C05358=1027.695,418.842,-151.802,174.340,48.612,159.982
C05359=1027.684,418.597,-151.753,174.327,48.608,159.979
C05360=1027.673,418.352,-151.706,174.314,48.605,159.976
C05361=1027.662,418.107,-151.658,174.301,48.601,159.973
C05362=1027.651,417.862,-151.609,174.288,48.597,159.971
C05363=1027.639,417.616,-151.562,174.275,48.593,159.967
C05364=1027.628,417.372,-151.514,174.262,48.590,159.965
C05365=1027.617,417.126,-151.467,174.249,48.586,159.962
C05366=1027.606,416.881,-151.418,174.236,48.583,159.959
C05367=1027.595,416.636,-151.370,174.223,48.579,159.956
C05368=1027.584,416.390,-151.323,174.210,48.576,159.953
C05369=1027.573,416.145,-151.275,174.197,48.572,159.950
C05370=1027.562,415.900,-151.229,174.184,48.569,159.947
C05371=1027.550,415.655,-151.181,174.171,48.565,159.944
C05372=1027.539,415.409,-151.133,174.160,48.562,159.942
C05373=1027.528,415.164,-151.087,174.147,48.558,159.939
C05374=1027.517,414.918,-151.040,174.134,48.555,159.936
C05375=1027.506,414.674,-150.992,174.121,48.551,159.933
C05376=1027.495,414.428,-150.945,174.108,48.548,159.930
C05377=1027.484,414.183,-150.898,174.097,48.545,159.928
C05378=1027.473,413.937,-150.851,174.084,48.541,159.925
C05379=1027.462,413.692,-150.804,174.071,48.538,159.922
C05380=1027.450,413.446,-150.757,174.060,48.535,159.919
C05381=1027.440,413.201,-150.710,174.047,48.531,159.917
C05382=1027.429,412.956,-150.663,174.034,48.528,159.914
C05383=1027.418,412.711,-150.616,174.022,48.524,159.911
C05384=1027.407,412.465,-150.569,174.010,48.522,159.908
C05385=1027.397,412.220,-150.523,173.998,48.518,159.906
C05386=1027.386,411.975,-150.476,173.986,48.515,159.903
C05387=1027.376,411.729,-150.429,173.974,48.512,159.900
C05388=1027.364,411.484,-150.382,173.962,48.509,159.898
C05389=1027.354,411.238,-150.336,173.950,48.505,159.895
C05390=1027.343,410.993,-150.289,173.937,48.502,159.892
C05391=1027.333,410.747,-150.243,173.926,48.499,159.890
C05392=1027.322,410.502,-150.197,173.913,48.496,159.887
C05393=1027.309,410.210,-150.141,173.899,48.492,159.884
C05394=1027.297,409.918,-150.086,173.885,48.488,159.881
C05395=1027.284,409.626,-150.031,173.871,48.484,159.878
C05396=1027.271,409.334,-149.976,173.857,48.481,159.875
C05397=1027.261,409.088,-149.930,173.846,48.478,159.872
C05398=1027.250,408.842,-149.884,173.834,48.475,159.870
C05399=1027.240,408.597,-149.838,173.822,48.472,159.867
C05400=1027.229,408.351,-149.792,173.810,48.469,159.865
C05401=1027.218,408.106,-149.746,173.799,48.466,159.862
C05402=1027.208,407.860,-149.700,173.788,48.463,159.860
C05403=1027.197,407.615,-149.655,173.775,48.460,159.857
C05404=1027.186,407.370,-149.610,173.764,48.458,159.855
C05405=1027.176,407.124,-149.564,173.753,48.454,159.852
C05406=1027.165,406.879,-149.518,173.742,48.452,159.850
C05407=1027.155,406.632,-149.473,173.729,48.449,159.847
C05408=1027.145,406.387,-149.427,173.718,48.446,159.845
C05409=1027.134,406.142,-149.381,173.707,48.443,159.843
C05410=1027.123,405.896,-149.335,173.696,48.440,159.840
C05411=1027.113,405.650,-149.290,173.684,48.437,159.838
C05412=1027.103,405.405,-149.244,173.673,48.434,159.835
C05413=1027.093,405.159,-149.199,173.662,48.432,159.833
C05414=1027.083,404.914,-149.154,173.651,48.429,159.831
C05415=1027.072,404.668,-149.109,173.640,48.426,159.828
C05416=1027.062,404.422,-149.063,173.629,48.423,159.826
C05417=1027.052,404.177,-149.018,173.618,48.421,159.824
C05418=1027.042,403.931,-148.972,173.607,48.418,159.821
C05419=1027.032,403.686,-148.927,173.595,48.415,159.819
C05420=1027.021,403.439,-148.882,173.584,48.413,159.817
C05421=1027.012,403.194,-148.837,173.573,48.410,159.814
C05422=1027.002,402.949,-148.792,173.562,48.407,159.812
C05423=1026.991,402.703,-148.746,173.551,48.404,159.810
C05424=1026.982,402.457,-148.702,173.540,48.402,159.807
C05425=1026.972,402.212,-148.657,173.529,48.399,159.805
C05426=1026.962,401.966,-148.612,173.518,48.397,159.803
C05427=1026.952,401.720,-148.567,173.508,48.394,159.801
C05428=1026.942,401.475,-148.522,173.497,48.391,159.798
C05429=1026.931,401.229,-148.477,173.486,48.389,159.796
C05430=1026.921,400.983,-148.432,173.475,48.386,159.794
C05431=1026.912,400.738,-148.388,173.465,48.384,159.792
C05432=1026.902,400.492,-148.343,173.453,48.381,159.789
C05433=1026.892,400.246,-148.298,173.444,48.379,159.787
C05434=1026.882,400.000,-148.254,173.433,48.376,159.785
C05435=1026.872,399.755,-148.209,173.422,48.374,159.783
C05436=1026.862,399.509,-148.164,173.411,48.372,159.781
C05437=1026.853,399.263,-148.120,173.401,48.369,159.778
C05438=1026.842,399.018,-148.076,173.390,48.367,159.776
C05439=1026.833,398.772,-148.032,173.379,48.364,159.774
C05440=1026.823,398.525,-147.987,173.370,48.362,159.772
C05441=1026.812,398.280,-147.943,173.359,48.360,159.770
C05442=1026.803,398.034,-147.898,173.348,48.357,159.768
C05443=1026.793,397.788,-147.855,173.338,48.355,159.765
C05444=1026.783,397.542,-147.811,173.328,48.353,159.763
C05445=1026.774,397.296,-147.767,173.317,48.350,159.761
C05446=1026.763,397.051,-147.723,173.307,48.348,159.759
C05447=1026.754,396.805,-147.678,173.296,48.346,159.757
C05448=1026.744,396.559,-147.635,173.287,48.343,159.755
C05449=1026.734,396.313,-147.591,173.276,48.342,159.753
C05450=1026.724,396.067,-147.547,173.266,48.339,159.751
C05451=1026.715,395.821,-147.504,173.256,48.337,159.749
C05452=1026.705,395.576,-147.460,173.246,48.334,159.747
C05453=1026.695,395.306,-147.412,173.234,48.332,159.744
C05454=1026.684,395.034,-147.363,173.223,48.330,159.742
C05455=1026.674,394.765,-147.315,173.212,48.327,159.740
C05456=1026.663,394.495,-147.267,173.202,48.325,159.738
C05457=1026.653,394.249,-147.224,173.191,48.323,159.736
C05458=1026.645,394.003,-147.180,173.181,48.321,159.734
C05459=1026.634,393.757,-147.137,173.171,48.319,159.732
C05460=1026.625,393.511,-147.093,173.161,48.317,159.730
C05461=1026.615,393.265,-147.050,173.152,48.315,159.728
C05462=1026.606,393.019,-147.006,173.141,48.312,159.726
C05463=1026.597,392.773,-146.963,173.132,48.310,159.724
C05464=1026.586,392.527,-146.920,173.121,48.309,159.722
C05465=1026.578,392.281,-146.877,173.112,48.307,159.720
C05466=1026.568,392.035,-146.833,173.102,48.304,159.718
C05467=1026.558,391.789,-146.791,173.092,48.303,159.716
C05468=1026.549,391.543,-146.747,173.082,48.301,159.714
C05469=1026.539,391.297,-146.704,173.073,48.299,159.712
C05470=1026.530,391.051,-146.662,173.063,48.297,159.711
C05471=1026.521,390.805,-146.618,173.053,48.295,159.709
C05472=1026.511,390.559,-146.575,173.044,48.293,159.707
C05473=1026.502,390.312,-146.532,173.034,48.291,159.705
C05474=1026.493,390.067,-146.489,173.024,48.289,159.703
C05475=1026.483,389.821,-146.446,173.014,48.287,159.701
C05476=1026.474,389.575,-146.403,173.005,48.285,159.699
C05477=1026.465,389.329,-146.360,172.996,48.283,159.697
C05478=1026.455,389.083,-146.317,172.987,48.282,159.696
C05479=1026.446,388.837,-146.275,172.976,48.280,159.694
C05480=1026.437,388.590,-146.232,172.967,48.278,159.692
C05481=1026.428,388.344,-146.189,172.957,48.276,159.690
C05482=1026.418,388.097,-146.147,172.948,48.275,159.688
C05483=1026.409,387.852,-146.105,172.939,48.273,159.686
C05484=1026.400,387.606,-146.062,172.930,48.271,159.685
C05485=1026.391,387.360,-146.019,172.920,48.269,159.683
C05486=1026.381,387.113,-145.976,172.910,48.268,159.681
C05487=1026.372,386.867,-145.935,172.901,48.266,159.679
C05488=1026.363,386.621,-145.892,172.892,48.264,159.677
C05489=1026.354,386.376,-145.850,172.883,48.263,159.676
C05490=1026.344,386.128,-145.808,172.873,48.261,159.674
C05491=1026.335,385.883,-145.765,172.864,48.259,159.672
C05492=1026.326,385.636,-145.724,172.855,48.258,159.671
C05493=1026.317,385.391,-145.681,172.846,48.256,159.669
C05494=1026.307,385.144,-145.639,172.837,48.255,159.667
C05495=1026.299,384.897,-145.597,172.828,48.253,159.665
C05496=1026.289,384.651,-145.555,172.818,48.252,159.664
C05497=1026.280,384.405,-145.513,172.809,48.250,159.662
C05498=1026.271,384.159,-145.472,172.800,48.248,159.660
C05499=1026.262,383.913,-145.429,172.791,48.247,159.659
C05500=1026.253,383.667,-145.387,172.782,48.245,159.657
C05501=1026.244,383.420,-145.346,172.773,48.244,159.655
C05502=1026.235,383.174,-145.304,172.764,48.242,159.654
C05503=1026.226,382.927,-145.262,172.755,48.241,159.652
C05504=1026.218,382.681,-145.221,172.746,48.240,159.650
C05505=1026.209,382.435,-145.179,172.737,48.238,159.649
C05506=1026.199,382.189,-145.138,172.728,48.237,159.647
C05507=1026.190,381.942,-145.096,172.719,48.235,159.645
C05508=1026.181,381.696,-145.054,172.710,48.234,159.644
C05509=1026.172,381.456,-145.013,172.702,48.233,159.642
C05510=1026.163,381.216,-144.972,172.693,48.231,159.641
C05511=1026.155,380.976,-144.932,172.684,48.230,159.639
C05512=1026.146,380.736,-144.891,172.676,48.229,159.638
C05513=1026.138,380.496,-144.851,172.667,48.227,159.636
C05514=1026.129,380.257,-144.811,172.659,48.226,159.634
C05515=1026.120,380.017,-144.770,172.650,48.225,159.633
C05516=1026.112,379.776,-144.730,172.641,48.223,159.631
C05517=1026.104,379.530,-144.689,172.632,48.222,159.630
C05518=1026.095,379.284,-144.647,172.624,48.220,159.628
C05519=1026.086,379.037,-144.606,172.616,48.220,159.627
C05520=1026.077,378.790,-144.565,172.607,48.218,159.625
C05521=1026.068,378.545,-144.524,172.598,48.217,159.623
C05522=1026.059,378.298,-144.483,172.590,48.216,159.622
C05523=1026.051,378.052,-144.441,172.581,48.214,159.620
C05524=1026.042,377.805,-144.400,172.572,48.213,159.619
C05525=1026.034,377.559,-144.359,172.564,48.212,159.617
C05526=1026.025,377.312,-144.318,172.555,48.211,159.616
C05527=1026.017,377.066,-144.276,172.547,48.210,159.614
C05528=1026.008,376.819,-144.235,172.539,48.208,159.613
C05529=1025.999,376.573,-144.195,172.530,48.207,159.611
C05530=1025.990,376.327,-144.154,172.521,48.206,159.610
C05531=1025.982,376.080,-144.113,172.512,48.205,159.608
C05532=1025.972,375.833,-144.072,172.505,48.204,159.607
C05533=1025.964,375.587,-144.032,172.496,48.203,159.605
C05534=1025.955,375.340,-143.991,172.488,48.201,159.604
C05535=1025.947,375.094,-143.951,172.479,48.201,159.602
C05536=1025.937,374.847,-143.910,172.470,48.200,159.601
C05537=1025.929,374.601,-143.869,172.463,48.199,159.600
C05538=1025.921,374.354,-143.828,172.454,48.198,159.598
C05539=1025.912,374.108,-143.788,172.445,48.197,159.597
C05540=1025.903,373.861,-143.747,172.438,48.196,159.595
C05541=1025.895,373.615,-143.707,172.429,48.195,159.594
C05542=1025.886,373.368,-143.666,172.421,48.193,159.592
C05543=1025.877,373.122,-143.626,172.413,48.193,159.591
C05544=1025.869,372.875,-143.585,172.405,48.191,159.589
C05545=1025.861,372.628,-143.545,172.396,48.191,159.588
C05546=1025.852,372.382,-143.505,172.388,48.190,159.587
C05547=1025.844,372.135,-143.464,172.380,48.189,159.585
C05548=1025.835,371.889,-143.424,172.371,48.188,159.584
C05549=1025.827,371.642,-143.384,172.364,48.187,159.583
C05550=1025.818,371.396,-143.344,172.355,48.187,159.581
C05551=1025.810,371.149,-143.303,172.348,48.185,159.580
C05552=1025.802,370.903,-143.263,172.340,48.184,159.578
C05553=1025.793,370.656,-143.223,172.331,48.184,159.577
C05554=1025.785,370.409,-143.183,172.324,48.183,159.576
C05555=1025.776,370.163,-143.143,172.315,48.182,159.574
C05556=1025.768,369.916,-143.103,172.308,48.181,159.573
C05557=1025.760,369.670,-143.063,172.299,48.180,159.572
C05558=1025.751,369.423,-143.023,172.292,48.180,159.571
C05559=1025.743,369.176,-142.982,172.283,48.179,159.569
C05560=1025.735,368.930,-142.943,172.276,48.178,159.568
C05561=1025.727,368.683,-142.903,172.268,48.177,159.566
C05562=1025.718,368.437,-142.863,172.259,48.177,159.565
C05563=1025.710,368.190,-142.824,172.252,48.176,159.564
C05564=1025.701,367.943,-142.784,172.243,48.175,159.563
C05565=1025.693,367.696,-142.744,172.236,48.175,159.561
C05566=1025.685,367.449,-142.705,172.228,48.173,159.560
C05567=1025.676,367.203,-142.665,172.220,48.173,159.559
C05568=1025.668,366.956,-142.626,172.213,48.173,159.558
C05569=1025.660,366.727,-142.589,172.205,48.172,159.556
C05570=1025.652,366.498,-142.552,172.198,48.171,159.555
C05571=1025.645,366.269,-142.515,172.190,48.171,159.554
C05572=1025.637,366.039,-142.479,172.183,48.170,159.553
C05573=1025.629,365.809,-142.442,172.176,48.170,159.552
C05574=1025.622,365.580,-142.405,172.169,48.170,159.551
C05575=1025.614,365.351,-142.369,172.162,48.169,159.549
C05576=1025.607,365.122,-142.332,172.155,48.168,159.548
C05577=1025.598,364.875,-142.293,172.147,48.168,159.547
C05578=1025.590,364.629,-142.253,172.139,48.167,159.546
C05579=1025.582,364.381,-142.215,172.132,48.166,159.545
C05580=1025.573,364.135,-142.175,172.124,48.166,159.543
C05581=1025.566,363.888,-142.136,172.116,48.166,159.542
C05582=1025.557,363.641,-142.096,172.109,48.165,159.541
C05583=1025.549,363.394,-142.058,172.101,48.164,159.540
C05584=1025.540,363.147,-142.018,172.094,48.164,159.539
C05585=1025.533,362.901,-141.978,172.086,48.163,159.537
C05586=1025.525,362.654,-141.940,172.079,48.163,159.536
C05587=1025.517,362.407,-141.901,172.071,48.163,159.535
C05588=1025.509,362.160,-141.862,172.064,48.162,159.534
C05589=1025.500,361.914,-141.823,172.056,48.161,159.533
C05590=1025.493,361.666,-141.784,172.048,48.161,159.531
C05591=1025.485,361.420,-141.745,172.041,48.161,159.530
C05592=1025.477,361.173,-141.706,172.034,48.160,159.529
C05593=1025.468,360.926,-141.667,172.026,48.160,159.528
C05594=1025.460,360.679,-141.628,172.019,48.159,159.527
C05595=1025.453,360.433,-141.589,172.012,48.159,159.526
C05596=1025.445,360.186,-141.550,172.004,48.159,159.525
C05597=1025.437,359.939,-141.511,171.997,48.159,159.524
C05598=1025.428,359.691,-141.473,171.989,48.158,159.522
C05599=1025.421,359.445,-141.434,171.982,48.158,159.521
C05600=1025.412,359.198,-141.395,171.975,48.158,159.520
C05601=1025.404,358.951,-141.357,171.968,48.158,159.519
C05602=1025.397,358.705,-141.318,171.959,48.157,159.518
C05603=1025.388,358.458,-141.280,171.952,48.157,159.517
C05604=1025.380,358.210,-141.242,171.945,48.157,159.516
C05605=1025.372,357.964,-141.204,171.938,48.157,159.515
C05606=1025.364,357.717,-141.165,171.931,48.157,159.514
C05607=1025.356,357.470,-141.127,171.924,48.156,159.513
C05608=1025.348,357.223,-141.088,171.916,48.156,159.512
C05609=1025.340,356.976,-141.049,171.909,48.156,159.511
C05610=1025.333,356.729,-141.011,171.902,48.155,159.509
C05611=1025.324,356.482,-140.973,171.895,48.155,159.508
C05612=1025.317,356.235,-140.934,171.888,48.155,159.507
C05613=1025.308,355.989,-140.896,171.880,48.155,159.506
C05614=1025.301,355.741,-140.859,171.873,48.155,159.505
C05615=1025.293,355.494,-140.820,171.866,48.155,159.504
C05616=1025.285,355.248,-140.782,171.859,48.155,159.503
C05617=1025.277,355.000,-140.743,171.852,48.155,159.502
C05618=1025.270,354.753,-140.706,171.844,48.155,159.501
C05619=1025.262,354.506,-140.667,171.837,48.155,159.500
C05620=1025.253,354.260,-140.630,171.830,48.155,159.499
C05621=1025.246,354.013,-140.592,171.823,48.155,159.498
C05622=1025.238,353.766,-140.553,171.816,48.155,159.497
C05623=1025.230,353.519,-140.516,171.809,48.155,159.496
C05624=1025.222,353.272,-140.478,171.802,48.155,159.495
C05625=1025.214,353.024,-140.440,171.795,48.154,159.494
C05626=1025.206,352.778,-140.403,171.788,48.154,159.493
C05627=1025.198,352.530,-140.365,171.781,48.154,159.492
C05628=1025.191,352.284,-140.327,171.774,48.154,159.491
C05629=1025.183,352.058,-140.292,171.768,48.155,159.490
C05630=1025.176,351.832,-140.258,171.761,48.155,159.489
C05631=1025.170,351.606,-140.223,171.755,48.154,159.488
C05632=1025.162,351.380,-140.189,171.749,48.155,159.488
C05633=1025.155,351.154,-140.154,171.743,48.155,159.487
C05634=1025.147,350.928,-140.120,171.737,48.155,159.486
C05635=1025.141,350.702,-140.086,171.730,48.155,159.485
C05636=1025.134,350.476,-140.051,171.724,48.155,159.484
C05637=1025.126,350.229,-140.014,171.717,48.155,159.483
C05638=1025.119,349.982,-139.976,171.710,48.155,159.482
C05639=1025.111,349.734,-139.939,171.704,48.156,159.481
C05640=1025.103,349.488,-139.901,171.696,48.156,159.480
C05641=1025.096,349.241,-139.863,171.689,48.155,159.479
C05642=1025.088,348.993,-139.826,171.683,48.156,159.479
C05643=1025.080,348.747,-139.789,171.676,48.156,159.478
C05644=1025.073,348.499,-139.751,171.670,48.156,159.477
C05645=1025.065,348.252,-139.714,171.663,48.156,159.476
C05646=1025.057,348.005,-139.677,171.656,48.156,159.475
C05647=1025.050,347.758,-139.639,171.649,48.157,159.474
C05648=1025.042,347.511,-139.602,171.642,48.157,159.473
C05649=1025.035,347.264,-139.565,171.636,48.157,159.472
C05650=1025.027,347.017,-139.528,171.629,48.158,159.471
C05651=1025.019,346.769,-139.491,171.622,48.158,159.470
C05652=1025.012,346.522,-139.454,171.616,48.158,159.470
C05653=1025.004,346.275,-139.417,171.609,48.158,159.469
C05654=1024.997,346.028,-139.379,171.602,48.159,159.468
C05655=1024.988,345.781,-139.342,171.596,48.159,159.467
C05656=1024.981,345.533,-139.305,171.589,48.159,159.466
C05657=1024.973,345.286,-139.268,171.582,48.160,159.465
C05658=1024.965,345.039,-139.232,171.576,48.160,159.465
C05659=1024.958,344.792,-139.195,171.570,48.161,159.464
C05660=1024.950,344.545,-139.158,171.562,48.161,159.463
C05661=1024.943,344.297,-139.121,171.556,48.161,159.462
C05662=1024.936,344.051,-139.084,171.549,48.162,159.461
C05663=1024.928,343.804,-139.047,171.543,48.162,159.460
C05664=1024.921,343.556,-139.011,171.537,48.163,159.460
C05665=1024.913,343.310,-138.974,171.530,48.162,159.459
C05666=1024.905,343.062,-138.937,171.523,48.163,159.458
C05667=1024.898,342.815,-138.900,171.517,48.163,159.457
C05668=1024.890,342.567,-138.864,171.511,48.164,159.456
C05669=1024.883,342.320,-138.828,171.504,48.164,159.455
C05670=1024.876,342.073,-138.790,171.497,48.165,159.455
C05671=1024.868,341.825,-138.754,171.491,48.165,159.454
C05672=1024.860,341.579,-138.717,171.485,48.166,159.453
C05673=1024.854,341.332,-138.680,171.478,48.166,159.452
C05674=1024.846,341.084,-138.644,171.471,48.167,159.451
C05675=1024.838,340.837,-138.608,171.466,48.167,159.451
C05676=1024.831,340.590,-138.570,171.459,48.168,159.450
C05677=1024.824,340.343,-138.535,171.452,48.168,159.449
C05678=1024.816,340.095,-138.498,171.446,48.169,159.448
C05679=1024.809,339.848,-138.462,171.440,48.169,159.448
C05680=1024.802,339.600,-138.425,171.433,48.170,159.447
C05681=1024.794,339.353,-138.388,171.427,48.171,159.446
C05682=1024.787,339.107,-138.353,171.421,48.171,159.445
C05683=1024.779,338.859,-138.316,171.414,48.172,159.445
C05684=1024.771,338.612,-138.280,171.408,48.172,159.444
C05685=1024.764,338.365,-138.244,171.401,48.173,159.443
C05686=1024.756,338.118,-138.208,171.396,48.174,159.442
C05687=1024.749,337.870,-138.172,171.389,48.174,159.442
C05688=1024.741,337.622,-138.136,171.383,48.176,159.441
C05689=1024.735,337.395,-138.102,171.377,48.176,159.440
C05690=1024.728,337.168,-138.070,171.372,48.177,159.440
C05691=1024.721,336.940,-138.036,171.366,48.177,159.439
C05692=1024.714,336.713,-138.003,171.359,48.178,159.438
C05693=1024.708,336.485,-137.970,171.354,48.178,159.438
C05694=1024.700,336.257,-137.937,171.348,48.179,159.437
C05695=1024.694,336.030,-137.904,171.343,48.179,159.436
C05696=1024.687,335.803,-137.871,171.337,48.180,159.436
C05697=1024.680,335.555,-137.836,171.331,48.181,159.435
C05698=1024.673,335.307,-137.799,171.324,48.182,159.434
C05699=1024.666,335.061,-137.763,171.319,48.182,159.434
C05700=1024.658,334.813,-137.727,171.312,48.184,159.433
C05701=1024.651,334.565,-137.691,171.306,48.184,159.432
C05702=1024.644,334.318,-137.656,171.300,48.185,159.432
C05703=1024.636,334.071,-137.619,171.293,48.186,159.431
C05704=1024.629,333.824,-137.584,171.288,48.186,159.430
C05705=1024.622,333.576,-137.548,171.281,48.187,159.429
C05706=1024.615,333.329,-137.513,171.275,48.188,159.429
C05707=1024.607,333.081,-137.477,171.270,48.189,159.428
C05708=1024.600,332.834,-137.442,171.263,48.190,159.427
C05709=1024.592,332.587,-137.406,171.258,48.190,159.427
C05710=1024.585,332.340,-137.371,171.251,48.192,159.426
C05711=1024.578,332.093,-137.335,171.245,48.193,159.426
C05712=1024.571,331.845,-137.299,171.239,48.193,159.425
C05713=1024.563,331.598,-137.265,171.233,48.194,159.424
C05714=1024.556,331.350,-137.229,171.227,48.195,159.424
C05715=1024.549,331.103,-137.194,171.221,48.196,159.423
C05716=1024.542,330.855,-137.158,171.215,48.198,159.423
C05717=1024.535,330.607,-137.123,171.209,48.198,159.422
C05718=1024.527,330.361,-137.088,171.203,48.199,159.421
C05719=1024.520,330.113,-137.052,171.197,48.200,159.421
C05720=1024.513,329.866,-137.017,171.191,48.201,159.420
C05721=1024.506,329.618,-136.982,171.185,48.202,159.419
C05722=1024.498,329.371,-136.946,171.179,48.203,159.419
C05723=1024.491,329.124,-136.911,171.174,48.204,159.418
C05724=1024.484,328.876,-136.876,171.167,48.205,159.418
C05725=1024.477,328.628,-136.840,171.161,48.206,159.417
C05726=1024.470,328.381,-136.805,171.156,48.207,159.416
C05727=1024.463,328.134,-136.771,171.149,48.208,159.416
C05728=1024.456,327.886,-136.736,171.144,48.209,159.415
C05729=1024.448,327.638,-136.700,171.138,48.210,159.415
C05730=1024.441,327.392,-136.664,171.132,48.211,159.414
C05731=1024.435,327.144,-136.629,171.126,48.212,159.414
C05732=1024.427,326.897,-136.595,171.120,48.213,159.413
C05733=1024.419,326.649,-136.560,171.114,48.215,159.412
C05734=1024.412,326.401,-136.525,171.109,48.215,159.412
C05735=1024.405,326.154,-136.491,171.103,48.217,159.411
C05736=1024.397,325.907,-136.456,171.097,48.218,159.411
C05737=1024.390,325.659,-136.421,171.091,48.219,159.410
C05738=1024.383,325.412,-136.387,171.085,48.220,159.410
C05739=1024.375,325.165,-136.352,171.079,48.222,159.409
C05740=1024.369,324.917,-136.318,171.073,48.223,159.409
C05741=1024.361,324.670,-136.283,171.068,48.224,159.408
C05742=1024.353,324.422,-136.248,171.062,48.226,159.408
C05743=1024.347,324.174,-136.214,171.056,48.227,159.407
C05744=1024.339,323.927,-136.180,171.050,48.228,159.406
C05745=1024.332,323.680,-136.145,171.045,48.229,159.406
C05746=1024.325,323.432,-136.111,171.039,48.231,159.405
C05747=1024.318,323.185,-136.076,171.034,48.232,159.405
C05748=1024.311,322.937,-136.042,171.027,48.233,159.404
C05749=1024.304,322.707,-136.010,171.022,48.235,159.404
C05750=1024.297,322.477,-135.977,171.017,48.236,159.404
C05751=1024.290,322.248,-135.946,171.011,48.237,159.403
C05752=1024.284,322.018,-135.914,171.006,48.238,159.403
C05753=1024.277,321.788,-135.881,171.001,48.240,159.402
C05754=1024.270,321.558,-135.850,170.996,48.240,159.402
C05755=1024.264,321.328,-135.818,170.991,48.242,159.401
C05756=1024.258,321.099,-135.786,170.986,48.243,159.401
C05757=1024.251,320.851,-135.752,170.980,48.245,159.400
C05758=1024.243,320.604,-135.718,170.974,48.245,159.400
C05759=1024.236,320.356,-135.684,170.968,48.247,159.399
C05760=1024.230,320.108,-135.649,170.963,48.248,159.399
C05761=1024.222,319.861,-135.615,170.957,48.250,159.398
C05762=1024.215,319.614,-135.581,170.952,48.251,159.398
C05763=1024.208,319.366,-135.547,170.946,48.252,159.397
C05764=1024.201,319.118,-135.512,170.940,48.254,159.397
C05765=1024.194,318.871,-135.478,170.935,48.256,159.397
C05766=1024.187,318.623,-135.444,170.929,48.257,159.396
C05767=1024.180,318.375,-135.410,170.924,48.258,159.396
C05768=1024.173,318.129,-135.376,170.918,48.260,159.395
C05769=1024.167,317.881,-135.341,170.912,48.261,159.395
C05770=1024.160,317.633,-135.307,170.907,48.263,159.394
C05771=1024.152,317.385,-135.274,170.901,48.264,159.394
C05772=1024.146,317.137,-135.239,170.896,48.265,159.393
C05773=1024.138,316.890,-135.205,170.890,48.267,159.393
C05774=1024.132,316.643,-135.171,170.885,48.269,159.393
C05775=1024.125,316.396,-135.137,170.880,48.270,159.392
C05776=1024.118,316.148,-135.103,170.874,48.271,159.392
C05777=1024.111,315.900,-135.069,170.868,48.273,159.391
C05778=1024.104,315.652,-135.035,170.863,48.274,159.391
C05779=1024.098,315.405,-135.001,170.857,48.276,159.390
C05780=1024.091,315.157,-134.967,170.852,48.278,159.390
C05781=1024.083,314.910,-134.934,170.846,48.279,159.390
C05782=1024.077,314.662,-134.899,170.841,48.281,159.389
C05783=1024.070,314.415,-134.866,170.836,48.282,159.389
C05784=1024.063,314.167,-134.832,170.830,48.284,159.388
C05785=1024.056,313.919,-134.798,170.825,48.285,159.388
C05786=1024.050,313.672,-134.764,170.820,48.287,159.387
C05787=1024.043,313.425,-134.730,170.814,48.288,159.387
C05788=1024.036,313.177,-134.696,170.809,48.290,159.387
C05789=1024.030,312.930,-134.662,170.804,48.291,159.386
C05790=1024.023,312.681,-134.629,170.798,48.293,159.386
C05791=1024.016,312.434,-134.596,170.793,48.295,159.385
C05792=1024.009,312.187,-134.562,170.788,48.296,159.385
C05793=1024.003,311.939,-134.528,170.783,48.298,159.385
C05794=1023.996,311.692,-134.494,170.777,48.299,159.384
C05795=1023.989,311.444,-134.460,170.771,48.301,159.384
C05796=1023.983,311.196,-134.428,170.766,48.302,159.384
C05797=1023.976,310.948,-134.393,170.760,48.304,159.383
C05798=1023.970,310.701,-134.360,170.755,48.306,159.383
C05799=1023.962,310.454,-134.326,170.750,48.307,159.382
C05800=1023.955,310.205,-134.293,170.744,48.309,159.382
C05801=1023.949,309.958,-134.260,170.740,48.311,159.382
C05802=1023.941,309.711,-134.227,170.735,48.313,159.381
C05803=1023.935,309.463,-134.194,170.728,48.315,159.381
C05804=1023.928,309.215,-134.160,170.724,48.317,159.381
C05805=1023.920,308.967,-134.128,170.718,48.319,159.380
C05806=1023.914,308.720,-134.095,170.713,48.321,159.380
C05807=1023.907,308.472,-134.061,170.708,48.322,159.380
C05808=1023.900,308.225,-134.029,170.702,48.324,159.379
C05809=1023.893,307.997,-133.999,170.697,48.326,159.379
C05810=1023.886,307.770,-133.968,170.693,48.327,159.379
C05811=1023.880,307.543,-133.938,170.689,48.330,159.379
C05812=1023.874,307.316,-133.908,170.684,48.331,159.378
C05813=1023.868,307.089,-133.878,170.678,48.333,159.378
C05814=1023.861,306.861,-133.848,170.674,48.335,159.378
C05815=1023.855,306.634,-133.817,170.669,48.336,159.377
C05816=1023.849,306.407,-133.787,170.664,48.338,159.377
C05817=1023.842,306.159,-133.754,170.659,48.340,159.377
C05818=1023.835,305.911,-133.722,170.654,48.342,159.377
C05819=1023.827,305.664,-133.688,170.648,48.344,159.376
C05820=1023.821,305.416,-133.655,170.644,48.346,159.376
C05821=1023.814,305.169,-133.623,170.639,48.347,159.376
C05822=1023.807,304.921,-133.590,170.633,48.350,159.375
C05823=1023.801,304.673,-133.557,170.628,48.352,159.375
C05824=1023.793,304.425,-133.525,170.623,48.354,159.375
C05825=1023.787,304.177,-133.492,170.617,48.356,159.375
C05826=1023.781,303.930,-133.459,170.612,48.357,159.374
C05827=1023.773,303.682,-133.427,170.608,48.360,159.374
C05828=1023.767,303.434,-133.394,170.602,48.362,159.374
C05829=1023.760,303.186,-133.361,170.597,48.364,159.373
C05830=1023.753,302.939,-133.329,170.592,48.366,159.373
C05831=1023.747,302.691,-133.296,170.587,48.368,159.373
C05832=1023.740,302.444,-133.264,170.581,48.370,159.373
C05833=1023.733,302.195,-133.231,170.577,48.372,159.372
C05834=1023.726,301.948,-133.198,170.572,48.374,159.372
C05835=1023.719,301.701,-133.166,170.567,48.376,159.372
C05836=1023.712,301.452,-133.133,170.561,48.378,159.372
C05837=1023.706,301.205,-133.100,170.557,48.380,159.371
C05838=1023.699,300.957,-133.068,170.552,48.382,159.371
C05839=1023.692,300.709,-133.035,170.547,48.384,159.371
C05840=1023.685,300.461,-133.003,170.541,48.386,159.371
C05841=1023.679,300.214,-132.971,170.536,48.388,159.370
C05842=1023.673,299.966,-132.938,170.532,48.391,159.370
C05843=1023.666,299.719,-132.906,170.527,48.393,159.370
C05844=1023.659,299.470,-132.873,170.521,48.394,159.370
C05845=1023.653,299.222,-132.841,170.516,48.397,159.369
C05846=1023.646,298.975,-132.809,170.512,48.399,159.369
C05847=1023.640,298.727,-132.776,170.507,48.401,159.369
C05848=1023.633,298.480,-132.744,170.501,48.403,159.369
C05849=1023.626,298.231,-132.711,170.496,48.406,159.369
C05850=1023.620,297.984,-132.679,170.492,48.408,159.368
C05851=1023.613,297.736,-132.646,170.487,48.409,159.368
C05852=1023.607,297.488,-132.614,170.482,48.411,159.368
C05853=1023.600,297.241,-132.582,170.476,48.414,159.368
C05854=1023.593,296.993,-132.549,170.472,48.416,159.367
C05855=1023.587,296.745,-132.517,170.467,48.418,159.367
C05856=1023.580,296.498,-132.485,170.462,48.420,159.367
C05857=1023.574,296.249,-132.453,170.458,48.422,159.367
C05858=1023.567,296.001,-132.420,170.452,48.425,159.367
C05859=1023.561,295.753,-132.389,170.447,48.427,159.366
C05860=1023.554,295.506,-132.356,170.442,48.429,159.366
C05861=1023.547,295.258,-132.324,170.438,48.431,159.366
C05862=1023.541,295.010,-132.292,170.433,48.433,159.366
C05863=1023.535,294.763,-132.259,170.427,48.436,159.366
C05864=1023.528,294.515,-132.228,170.423,48.438,159.365
C05865=1023.522,294.267,-132.196,170.418,48.440,159.365
C05866=1023.515,294.019,-132.163,170.413,48.442,159.365
C05867=1023.509,293.771,-132.131,170.408,48.445,159.365
C05868=1023.502,293.524,-132.099,170.404,48.447,159.365
C05869=1023.497,293.305,-132.071,170.399,48.450,159.365
C05870=1023.491,293.086,-132.043,170.395,48.452,159.365
C05871=1023.485,292.868,-132.015,170.391,48.454,159.364
C05872=1023.480,292.650,-131.987,170.386,48.456,159.364
C05873=1023.473,292.430,-131.959,170.383,48.458,159.364
C05874=1023.467,292.212,-131.931,170.378,48.460,159.364
C05875=1023.462,291.994,-131.903,170.373,48.462,159.364
C05876=1023.456,291.775,-131.876,170.370,48.464,159.364
C05877=1023.450,291.527,-131.844,170.365,48.467,159.364
C05878=1023.443,291.280,-131.812,170.359,48.469,159.363
C05879=1023.437,291.032,-131.780,170.355,48.471,159.363
C05880=1023.430,290.784,-131.749,170.350,48.474,159.363
C05881=1023.423,290.536,-131.717,170.346,48.476,159.363
C05882=1023.416,290.288,-131.686,170.341,48.478,159.363
C05883=1023.410,290.040,-131.654,170.336,48.481,159.363
C05884=1023.403,289.792,-131.623,170.331,48.483,159.363
C05885=1023.396,289.545,-131.591,170.327,48.486,159.363
C05886=1023.390,289.297,-131.560,170.322,48.488,159.362
C05887=1023.384,289.048,-131.528,170.317,48.491,159.362
C05888=1023.377,288.801,-131.497,170.312,48.494,159.362
C05889=1023.370,288.553,-131.465,170.307,48.497,159.362
C05890=1023.363,288.305,-131.434,170.303,48.499,159.362
C05891=1023.357,288.057,-131.402,170.298,48.501,159.362
C05892=1023.351,287.810,-131.371,170.294,48.504,159.362
C05893=1023.344,287.561,-131.341,170.288,48.507,159.362
C05894=1023.337,287.313,-131.309,170.284,48.509,159.361
C05895=1023.331,287.065,-131.278,170.279,48.512,159.361
C05896=1023.324,286.817,-131.246,170.275,48.514,159.361
C05897=1023.317,286.569,-131.215,170.270,48.517,159.361
C05898=1023.311,286.321,-131.184,170.265,48.519,159.361
C05899=1023.305,286.073,-131.152,170.260,48.522,159.361
C05900=1023.299,285.826,-131.121,170.256,48.525,159.361
C05901=1023.292,285.578,-131.090,170.251,48.527,159.361
C05902=1023.285,285.330,-131.058,170.247,48.530,159.361
C05903=1023.278,285.082,-131.028,170.242,48.533,159.361
C05904=1023.271,284.834,-130.997,170.237,48.535,159.361
C05905=1023.266,284.586,-130.966,170.232,48.538,159.361
C05906=1023.259,284.338,-130.935,170.228,48.541,159.361
C05907=1023.252,284.090,-130.903,170.223,48.543,159.361
C05908=1023.246,283.841,-130.873,170.219,48.546,159.360
C05909=1023.238,283.594,-130.842,170.214,48.548,159.360
C05910=1023.232,283.346,-130.811,170.209,48.552,159.360
C05911=1023.226,283.098,-130.780,170.205,48.554,159.360
C05912=1023.219,282.850,-130.749,170.200,48.557,159.360
C05913=1023.213,282.602,-130.718,170.196,48.559,159.360
C05914=1023.207,282.354,-130.688,170.191,48.562,159.360
C05915=1023.199,282.106,-130.657,170.186,48.565,159.360
C05916=1023.193,281.858,-130.626,170.182,48.568,159.360
C05917=1023.186,281.610,-130.595,170.177,48.571,159.360
C05918=1023.180,281.362,-130.564,170.173,48.574,159.360
C05919=1023.174,281.114,-130.533,170.168,48.576,159.360
C05920=1023.166,280.866,-130.503,170.164,48.579,159.360
C05921=1023.161,280.618,-130.472,170.158,48.582,159.360
C05922=1023.154,280.370,-130.441,170.154,48.585,159.360
C05923=1023.147,280.122,-130.410,170.150,48.587,159.360
C05924=1023.142,279.874,-130.380,170.145,48.590,159.360
C05925=1023.135,279.626,-130.348,170.141,48.593,159.360
C05926=1023.128,279.378,-130.318,170.137,48.596,159.360
C05927=1023.122,279.130,-130.288,170.132,48.599,159.360
C05928=1023.115,278.882,-130.256,170.127,48.602,159.360
C05929=1023.110,278.669,-130.230,170.123,48.604,159.360
C05930=1023.104,278.457,-130.204,170.120,48.606,159.360
C05931=1023.099,278.245,-130.178,170.115,48.609,159.360
C05932=1023.093,278.032,-130.152,170.112,48.611,159.360
C05933=1023.088,277.820,-130.125,170.108,48.614,159.360
C05934=1023.083,277.608,-130.099,170.104,48.616,159.359
C05935=1023.077,277.396,-130.073,170.101,48.619,159.360
C05936=1023.071,277.182,-130.047,170.096,48.621,159.360
C05937=1023.065,276.934,-130.016,170.092,48.624,159.360
C05938=1023.058,276.686,-129.986,170.088,48.627,159.360
C05939=1023.052,276.438,-129.956,170.083,48.630,159.360
C05940=1023.045,276.190,-129.926,170.079,48.633,159.360
C05941=1023.039,275.943,-129.895,170.074,48.637,159.360
C05942=1023.032,275.695,-129.865,170.069,48.639,159.360
C05943=1023.026,275.447,-129.834,170.065,48.642,159.360
C05944=1023.020,275.198,-129.803,170.061,48.645,159.360
C05945=1023.013,274.950,-129.773,170.056,48.648,159.360
C05946=1023.007,274.702,-129.743,170.052,48.651,159.360
C05947=1023.000,274.454,-129.713,170.047,48.654,159.360
C05948=1022.994,274.206,-129.683,170.043,48.657,159.360
C05949=1022.987,273.958,-129.653,170.038,48.660,159.360
C05950=1022.981,273.710,-129.623,170.034,48.664,159.360
C05951=1022.974,273.462,-129.593,170.030,48.666,159.360
C05952=1022.968,273.214,-129.562,170.026,48.669,159.360
C05953=1022.962,272.965,-129.532,170.021,48.672,159.360
C05954=1022.955,272.718,-129.502,170.016,48.676,159.360
C05955=1022.948,272.469,-129.472,170.012,48.679,159.360
C05956=1022.942,272.222,-129.441,170.007,48.681,159.360
C05957=1022.936,271.974,-129.412,170.003,48.685,159.360
C05958=1022.930,271.725,-129.382,169.999,48.688,159.360
C05959=1022.923,271.477,-129.352,169.995,48.691,159.360
C05960=1022.917,271.229,-129.321,169.991,48.694,159.360
C05961=1022.910,270.981,-129.291,169.985,48.697,159.360
C05962=1022.904,270.732,-129.261,169.981,48.701,159.360
C05963=1022.897,270.485,-129.232,169.977,48.703,159.360
C05964=1022.892,270.237,-129.201,169.973,48.707,159.361
C05965=1022.885,269.988,-129.172,169.969,48.710,159.361
C05966=1022.878,269.741,-129.142,169.965,48.713,159.361
C05967=1022.872,269.492,-129.111,169.960,48.716,159.361
C05968=1022.866,269.244,-129.082,169.955,48.720,159.361
C05969=1022.859,268.996,-129.053,169.951,48.723,159.361
C05970=1022.853,268.748,-129.022,169.947,48.726,159.361
C05971=1022.846,268.500,-128.993,169.942,48.729,159.361
C05972=1022.839,268.252,-128.963,169.938,48.732,159.361
C05973=1022.834,268.003,-128.933,169.934,48.735,159.361
C05974=1022.827,267.756,-128.903,169.930,48.739,159.361
C05975=1022.820,267.507,-128.874,169.925,48.743,159.361
C05976=1022.814,267.259,-128.844,169.921,48.745,159.361
C05977=1022.808,267.011,-128.815,169.917,48.749,159.362
C05978=1022.801,266.763,-128.784,169.912,48.752,159.362
C05979=1022.795,266.515,-128.755,169.908,48.755,159.362
C05980=1022.789,266.267,-128.725,169.904,48.759,159.362
C05981=1022.782,266.018,-128.696,169.900,48.762,159.362
C05982=1022.776,265.770,-128.666,169.895,48.765,159.362
C05983=1022.769,265.522,-128.637,169.891,48.769,159.362
C05984=1022.763,265.274,-128.608,169.887,48.772,159.362
C05985=1022.757,265.026,-128.577,169.882,48.775,159.362
C05986=1022.750,264.777,-128.548,169.878,48.779,159.362
C05987=1022.744,264.529,-128.519,169.874,48.782,159.363
C05988=1022.737,264.281,-128.489,169.869,48.786,159.363
C05989=1022.726,263.861,-128.440,169.863,48.791,159.363
C05990=1022.721,263.651,-128.415,169.859,48.794,159.363
C05991=1022.716,263.441,-128.390,169.855,48.797,159.363
C05992=1022.710,263.231,-128.365,169.852,48.800,159.363
C05993=1022.705,263.020,-128.340,169.848,48.803,159.363
C05994=1022.699,262.810,-128.315,169.845,48.806,159.363
C05995=1022.694,262.600,-128.291,169.842,48.809,159.364
C05996=1022.687,262.352,-128.261,169.836,48.812,159.364
C05997=1022.681,262.104,-128.232,169.832,48.815,159.364
C05998=1022.676,261.856,-128.202,169.828,48.819,159.364
C05999=1022.669,261.607,-128.173,169.824,48.822,159.364
C06000=1022.663,261.359,-128.144,169.820,48.826,159.364
C06001=1022.656,261.111,-128.114,169.816,48.829,159.364
C06002=1022.650,260.863,-128.085,169.812,48.833,159.365
C06003=1022.644,260.615,-128.056,169.808,48.836,159.365
C06004=1022.637,260.366,-128.027,169.803,48.840,159.365
C06005=1022.630,260.118,-127.998,169.799,48.844,159.365
C06006=1022.624,259.870,-127.968,169.795,48.847,159.365
C06007=1022.617,259.622,-127.940,169.791,48.851,159.365
C06008=1022.611,259.374,-127.911,169.787,48.854,159.366
C06009=1022.605,259.126,-127.882,169.782,48.858,159.366
C06010=1022.597,258.877,-127.854,169.778,48.861,159.366
C06011=1022.591,258.629,-127.825,169.774,48.865,159.366
C06012=1022.585,258.380,-127.796,169.770,48.869,159.366
C06013=1022.579,258.132,-127.767,169.766,48.873,159.367
C06014=1022.572,257.884,-127.738,169.761,48.876,159.367
C06015=1022.565,257.636,-127.709,169.757,48.880,159.367
C06016=1022.559,257.387,-127.681,169.753,48.883,159.367
C06017=1022.552,257.139,-127.652,169.749,48.887,159.367
C06018=1022.546,256.891,-127.623,169.746,48.891,159.368
C06019=1022.539,256.643,-127.594,169.741,48.895,159.368
C06020=1022.533,256.395,-127.565,169.737,48.898,159.368
C06021=1022.527,256.146,-127.537,169.733,48.902,159.368
C06022=1022.520,255.898,-127.508,169.729,48.906,159.368
C06023=1022.514,255.650,-127.479,169.725,48.910,159.369
C06024=1022.507,255.402,-127.451,169.720,48.913,159.369
C06025=1022.501,255.153,-127.422,169.716,48.917,159.369
C06026=1022.494,254.905,-127.393,169.712,48.921,159.369
C06027=1022.487,254.657,-127.365,169.708,48.925,159.369
C06028=1022.481,254.408,-127.336,169.704,48.928,159.370
C06029=1022.475,254.160,-127.307,169.701,48.932,159.370
C06030=1022.469,253.912,-127.278,169.696,48.936,159.370
C06031=1022.462,253.663,-127.250,169.692,48.940,159.370
C06032=1022.456,253.415,-127.221,169.688,48.943,159.370
C06033=1022.450,253.166,-127.193,169.684,48.947,159.371
C06034=1022.443,252.919,-127.165,169.680,48.951,159.371
C06035=1022.437,252.670,-127.136,169.675,48.955,159.371
C06036=1022.431,252.422,-127.107,169.671,48.959,159.371
C06037=1022.424,252.174,-127.079,169.667,48.962,159.371
C06038=1022.418,251.925,-127.050,169.664,48.966,159.372
C06039=1022.412,251.677,-127.021,169.660,48.970,159.372
C06040=1022.405,251.429,-126.994,169.656,48.973,159.372
C06041=1022.399,251.180,-126.965,169.651,48.978,159.372
C06042=1022.393,250.932,-126.936,169.647,48.981,159.373
C06043=1022.386,250.684,-126.907,169.643,48.986,159.373
C06044=1022.380,250.435,-126.880,169.639,48.989,159.373
C06045=1022.374,250.188,-126.851,169.636,48.993,159.374
C06046=1022.368,249.939,-126.823,169.632,48.997,159.374
C06047=1022.361,249.691,-126.794,169.628,49.000,159.374
C06048=1022.356,249.480,-126.770,169.624,49.004,159.374
C06049=1022.350,249.269,-126.746,169.621,49.007,159.374
C06050=1022.345,249.058,-126.721,169.617,49.011,159.374
C06051=1022.340,248.847,-126.698,169.614,49.014,159.375
C06052=1022.334,248.637,-126.673,169.611,49.017,159.375
C06053=1022.329,248.425,-126.650,169.607,49.021,159.375
C06054=1022.324,248.215,-126.625,169.604,49.024,159.375
C06055=1022.319,248.004,-126.602,169.601,49.027,159.376
C06056=1022.313,247.756,-126.573,169.596,49.031,159.376
C06057=1022.307,247.507,-126.544,169.592,49.035,159.376
C06058=1022.301,247.258,-126.516,169.588,49.039,159.376
C06059=1022.294,247.010,-126.487,169.584,49.043,159.377
C06060=1022.288,246.761,-126.459,169.581,49.047,159.377
C06061=1022.282,246.513,-126.431,169.577,49.050,159.377
C06062=1022.275,246.266,-126.403,169.573,49.055,159.377
C06063=1022.269,246.017,-126.374,169.568,49.059,159.378
C06064=1022.264,245.768,-126.346,169.564,49.063,159.378
C06065=1022.257,245.520,-126.318,169.561,49.067,159.378
C06066=1022.251,245.272,-126.289,169.557,49.070,159.378
C06067=1022.245,245.024,-126.261,169.553,49.074,159.379
C06068=1022.239,244.775,-126.234,169.549,49.079,159.379
C06069=1022.233,244.526,-126.205,169.545,49.082,159.379
C06070=1022.226,244.278,-126.176,169.541,49.087,159.380
C06071=1022.220,244.030,-126.149,169.537,49.090,159.380
C06072=1022.214,243.782,-126.121,169.533,49.094,159.380
C06073=1022.208,243.533,-126.092,169.530,49.099,159.380
C06074=1022.202,243.284,-126.064,169.526,49.103,159.381
C06075=1022.196,243.037,-126.037,169.522,49.106,159.381
C06076=1022.190,242.788,-126.009,169.518,49.110,159.381
C06077=1022.183,242.540,-125.980,169.514,49.115,159.382
C06078=1022.176,242.292,-125.953,169.510,49.119,159.382
C06079=1022.171,242.044,-125.925,169.506,49.123,159.382
C06080=1022.164,241.795,-125.897,169.502,49.127,159.382
C06081=1022.158,241.546,-125.869,169.499,49.131,159.383
C06082=1022.151,241.298,-125.841,169.494,49.136,159.383
C06083=1022.145,241.050,-125.813,169.490,49.140,159.383
C06084=1022.140,240.801,-125.786,169.487,49.144,159.384
C06085=1022.133,240.552,-125.758,169.483,49.148,159.384
C06086=1022.128,240.304,-125.730,169.479,49.152,159.385
C06087=1022.121,240.056,-125.702,169.475,49.156,159.385
C06088=1022.114,239.808,-125.675,169.471,49.160,159.385
C06089=1022.108,239.559,-125.646,169.467,49.165,159.385
C06090=1022.102,239.311,-125.619,169.463,49.169,159.386
C06091=1022.096,239.063,-125.591,169.460,49.173,159.386
C06092=1022.089,238.814,-125.564,169.456,49.177,159.386
C06093=1022.083,238.566,-125.537,169.452,49.182,159.387
C06094=1022.076,238.317,-125.509,169.448,49.186,159.387
C06095=1022.071,238.069,-125.481,169.445,49.191,159.388
C06096=1022.064,237.821,-125.454,169.441,49.195,159.388
C06097=1022.058,237.572,-125.427,169.436,49.199,159.388
C06098=1022.051,237.323,-125.399,169.433,49.204,159.389
C06099=1022.045,237.076,-125.371,169.429,49.208,159.389
C06100=1022.039,236.827,-125.344,169.425,49.212,159.389
C06101=1022.032,236.578,-125.317,169.421,49.217,159.390
C06102=1022.026,236.330,-125.289,169.417,49.221,159.390
C06103=1022.021,236.081,-125.262,169.413,49.225,159.390
C06104=1022.014,235.833,-125.234,169.410,49.230,159.391
C06105=1022.008,235.585,-125.207,169.407,49.234,159.391
C06106=1022.001,235.336,-125.180,169.402,49.239,159.391
C06107=1021.995,235.088,-125.152,169.398,49.243,159.392
C06108=1021.989,234.874,-125.129,169.396,49.247,159.392
C06109=1021.984,234.659,-125.105,169.392,49.250,159.392
C06110=1021.978,234.446,-125.082,169.389,49.254,159.393
C06111=1021.973,234.232,-125.058,169.385,49.258,159.393
C06112=1021.968,234.017,-125.034,169.381,49.262,159.393
C06113=1021.962,233.803,-125.011,169.379,49.266,159.394
C06114=1021.957,233.589,-124.988,169.375,49.269,159.394
C06115=1021.952,233.375,-124.965,169.372,49.273,159.394
C06116=1021.945,233.127,-124.937,169.369,49.277,159.395
C06117=1021.940,232.878,-124.910,169.365,49.282,159.395
C06118=1021.933,232.630,-124.882,169.361,49.287,159.396
C06119=1021.927,232.381,-124.855,169.357,49.291,159.396
C06120=1021.921,232.133,-124.828,169.353,49.295,159.396
C06121=1021.915,231.885,-124.801,169.350,49.300,159.397
C06122=1021.908,231.636,-124.773,169.345,49.305,159.397
C06123=1021.902,231.387,-124.746,169.342,49.309,159.397
C06124=1021.896,231.139,-124.719,169.339,49.314,159.398
C06125=1021.889,230.890,-124.692,169.335,49.318,159.398
C06126=1021.884,230.642,-124.665,169.330,49.323,159.399
C06127=1021.877,230.394,-124.637,169.327,49.327,159.399
C06128=1021.871,230.145,-124.611,169.323,49.332,159.399
C06129=1021.865,229.896,-124.584,169.320,49.337,159.400
C06130=1021.859,229.648,-124.556,169.315,49.341,159.400
C06131=1021.852,229.400,-124.530,169.312,49.345,159.401
C06132=1021.846,229.151,-124.503,169.309,49.350,159.401
C06133=1021.840,228.904,-124.476,169.305,49.354,159.402
C06134=1021.833,228.655,-124.449,169.301,49.360,159.402
C06135=1021.828,228.406,-124.422,169.297,49.364,159.402
C06136=1021.821,228.158,-124.395,169.294,49.369,159.403
C06137=1021.815,227.909,-124.368,169.290,49.373,159.403
C06138=1021.809,227.660,-124.341,169.286,49.378,159.404
C06139=1021.803,227.412,-124.314,169.282,49.382,159.404
C06140=1021.796,227.164,-124.287,169.279,49.387,159.405
C06141=1021.790,226.915,-124.260,169.275,49.392,159.405
C06142=1021.784,226.667,-124.234,169.271,49.397,159.405
C06143=1021.778,226.418,-124.207,169.267,49.401,159.406
C06144=1021.771,226.170,-124.181,169.264,49.406,159.406
C06145=1021.765,225.921,-124.154,169.260,49.411,159.407
C06146=1021.759,225.673,-124.127,169.256,49.415,159.407
C06147=1021.752,225.424,-124.101,169.253,49.420,159.408
C06148=1021.746,225.175,-124.074,169.249,49.425,159.408
C06149=1021.740,224.927,-124.048,169.245,49.430,159.408
C06150=1021.733,224.678,-124.021,169.242,49.435,159.409
C06151=1021.727,224.430,-123.994,169.239,49.439,159.410
C06152=1021.720,224.181,-123.968,169.234,49.445,159.410
C06153=1021.715,223.933,-123.941,169.231,49.449,159.410
C06154=1021.709,223.684,-123.915,169.227,49.454,159.411
C06155=1021.702,223.436,-123.888,169.223,49.459,159.411
C06156=1021.696,223.187,-123.861,169.219,49.463,159.412
C06157=1021.690,222.938,-123.834,169.216,49.468,159.412
C06158=1021.683,222.690,-123.808,169.212,49.473,159.413
C06159=1021.677,222.442,-123.782,169.209,49.478,159.413
C06160=1021.670,222.193,-123.755,169.205,49.483,159.414
C06161=1021.664,221.945,-123.729,169.201,49.488,159.414
C06162=1021.659,221.696,-123.702,169.198,49.493,159.415
C06163=1021.651,221.448,-123.676,169.194,49.498,159.415
C06164=1021.646,221.199,-123.649,169.191,49.503,159.416
C06165=1021.640,220.951,-123.622,169.186,49.507,159.416
C06166=1021.633,220.702,-123.596,169.183,49.512,159.416
C06167=1021.627,220.453,-123.570,169.180,49.517,159.417
C06168=1021.621,220.236,-123.547,169.176,49.521,159.417
C06169=1021.616,220.017,-123.524,169.173,49.526,159.418
C06170=1021.611,219.799,-123.500,169.170,49.530,159.418
C06171=1021.605,219.581,-123.477,169.167,49.534,159.419
C06172=1021.600,219.363,-123.453,169.163,49.538,159.419
C06173=1021.595,219.145,-123.430,169.161,49.543,159.420
C06174=1021.589,218.927,-123.408,169.157,49.547,159.420
C06175=1021.583,218.709,-123.384,169.154,49.552,159.420
C06176=1021.578,218.460,-123.358,169.150,49.556,159.421
C06177=1021.572,218.212,-123.332,169.147,49.561,159.421
C06178=1021.565,217.964,-123.306,169.143,49.567,159.422
C06179=1021.558,217.715,-123.280,169.140,49.572,159.422
C06180=1021.552,217.466,-123.254,169.136,49.576,159.423
C06181=1021.546,217.218,-123.228,169.132,49.582,159.423
C06182=1021.540,216.969,-123.202,169.129,49.587,159.424
C06183=1021.533,216.720,-123.175,169.125,49.592,159.424
C06184=1021.527,216.472,-123.149,169.122,49.597,159.425
C06185=1021.521,216.223,-123.123,169.119,49.602,159.426
C06186=1021.515,215.975,-123.097,169.114,49.608,159.426
C06187=1021.508,215.726,-123.071,169.111,49.613,159.427
C06188=1021.502,215.477,-123.045,169.108,49.617,159.427
C06189=1021.496,215.229,-123.019,169.104,49.623,159.428
C06190=1021.490,214.981,-122.993,169.100,49.628,159.428
C06191=1021.484,214.732,-122.967,169.096,49.633,159.429
C06192=1021.477,214.483,-122.941,169.093,49.638,159.429
C06193=1021.470,214.235,-122.915,169.090,49.643,159.430
C06194=1021.465,213.986,-122.889,169.086,49.649,159.430
C06195=1021.458,213.738,-122.863,169.082,49.654,159.431
C06196=1021.452,213.489,-122.838,169.079,49.659,159.431
C06197=1021.446,213.241,-122.812,169.075,49.664,159.432
C06198=1021.440,212.992,-122.785,169.072,49.669,159.432
C06199=1021.433,212.744,-122.759,169.068,49.675,159.433
C06200=1021.427,212.495,-122.734,169.065,49.680,159.434
C06201=1021.421,212.247,-122.707,169.061,49.685,159.434
C06202=1021.415,211.998,-122.682,169.057,49.690,159.435
C06203=1021.409,211.749,-122.657,169.054,49.695,159.435
C06204=1021.403,211.501,-122.630,169.050,49.701,159.436
C06205=1021.396,211.251,-122.604,169.047,49.706,159.436
C06206=1021.390,211.003,-122.578,169.044,49.711,159.437
C06207=1021.384,210.754,-122.552,169.039,49.716,159.437
C06208=1021.378,210.506,-122.526,169.036,49.721,159.438
C06209=1021.371,210.258,-122.501,169.033,49.726,159.439
C06210=1021.366,210.009,-122.475,169.029,49.732,159.439
C06211=1021.360,209.761,-122.449,169.026,49.737,159.440
C06212=1021.353,209.512,-122.424,169.022,49.742,159.440
C06213=1021.347,209.263,-122.398,169.019,49.747,159.441
C06214=1021.341,209.015,-122.373,169.015,49.753,159.441
C06215=1021.334,208.766,-122.346,169.011,49.758,159.442
C06216=1021.328,208.517,-122.321,169.009,49.764,159.443
C06217=1021.322,208.268,-122.295,169.004,49.769,159.443
C06218=1021.316,208.020,-122.270,169.001,49.774,159.444
C06219=1021.309,207.772,-122.244,168.997,49.780,159.444
C06220=1021.303,207.523,-122.218,168.994,49.785,159.445
C06221=1021.297,207.274,-122.193,168.990,49.791,159.445
C06222=1021.291,207.026,-122.168,168.987,49.796,159.446
C06223=1021.285,206.777,-122.142,168.984,49.802,159.447
C06224=1021.278,206.529,-122.116,168.980,49.807,159.447
C06225=1021.272,206.280,-122.091,168.977,49.812,159.448
C06226=1021.266,206.031,-122.066,168.973,49.818,159.448
C06227=1021.259,205.783,-122.040,168.970,49.823,159.449
C06228=1021.254,205.567,-122.018,168.967,49.828,159.450
C06229=1021.249,205.351,-121.996,168.963,49.833,159.450
C06230=1021.243,205.135,-121.974,168.961,49.837,159.451
C06231=1021.238,204.919,-121.952,168.958,49.842,159.451
C06232=1021.232,204.704,-121.930,168.954,49.847,159.452
C06233=1021.226,204.488,-121.908,168.951,49.852,159.452
C06234=1021.221,204.272,-121.886,168.948,49.857,159.453
C06235=1021.193,203.019,-121.765,168.506,49.767,159.362
C06236=1021.188,202.770,-121.742,168.502,49.773,159.363
C06237=1021.182,202.521,-121.718,168.497,49.780,159.364
C06238=1021.177,202.272,-121.694,168.492,49.786,159.364
C06239=1021.172,202.023,-121.670,168.489,49.793,159.365
C06240=1021.166,201.774,-121.647,168.484,49.799,159.365
C06241=1021.161,201.526,-121.623,168.480,49.805,159.366
C06242=1021.156,201.277,-121.599,168.475,49.812,159.367
C06243=1021.150,201.028,-121.575,168.472,49.818,159.367
C06244=1021.145,200.779,-121.552,168.467,49.825,159.368
C06245=1021.140,200.531,-121.528,168.462,49.831,159.369
C06246=1021.135,200.281,-121.504,168.458,49.838,159.369
C06247=1021.129,200.033,-121.480,168.454,49.844,159.370
C06248=1021.124,199.784,-121.457,168.450,49.851,159.371
C06249=1021.119,199.535,-121.433,168.445,49.857,159.371
C06250=1021.113,199.286,-121.410,168.442,49.864,159.372
C06251=1021.107,199.037,-121.387,168.437,49.871,159.373
C06252=1021.102,198.788,-121.363,168.432,49.877,159.373
C06253=1021.096,198.539,-121.340,168.429,49.884,159.374
C06254=1021.091,198.291,-121.316,168.424,49.890,159.374
C06255=1021.085,198.042,-121.293,168.419,49.897,159.375
C06256=1021.080,197.793,-121.270,168.416,49.904,159.376
C06257=1021.075,197.544,-121.246,168.411,49.910,159.376
C06258=1021.069,197.295,-121.224,168.407,49.917,159.377
C06259=1021.063,197.046,-121.201,168.403,49.924,159.378
C06260=1021.058,196.797,-121.176,168.399,49.930,159.379
C06261=1021.053,196.549,-121.154,168.394,49.937,159.379
C06262=1021.047,196.300,-121.131,168.390,49.944,159.380
C06263=1021.042,196.051,-121.107,168.386,49.950,159.381
C06264=1021.036,195.802,-121.084,168.381,49.957,159.381
C06265=1021.030,195.553,-121.061,168.378,49.963,159.382
C06266=1021.025,195.304,-121.038,168.373,49.970,159.383
C06267=1021.020,195.055,-121.015,168.369,49.976,159.383
C06268=1021.015,194.806,-120.991,168.365,49.983,159.384
C06269=1021.010,194.558,-120.969,168.360,49.990,159.385
C06270=1021.004,194.309,-120.946,168.356,49.996,159.385
C06271=1020.999,194.060,-120.922,168.352,50.003,159.386
C06272=1020.993,193.811,-120.899,168.348,50.010,159.387
C06273=1020.987,193.563,-120.876,168.343,50.016,159.387
C06274=1020.982,193.313,-120.852,168.340,50.023,159.388
C06275=1020.977,193.065,-120.830,168.335,50.030,159.389
C06276=1020.972,192.816,-120.807,168.331,50.036,159.389
C06277=1020.967,192.566,-120.784,168.327,50.043,159.390
C06278=1020.961,192.318,-120.761,168.323,50.050,159.391
C06279=1020.955,192.069,-120.738,168.318,50.056,159.391
C06280=1020.951,191.820,-120.715,168.315,50.063,159.392
C06281=1020.945,191.571,-120.692,168.310,50.070,159.393
C06282=1020.939,191.322,-120.669,168.307,50.076,159.394
C06283=1020.934,191.073,-120.645,168.302,50.083,159.394
C06284=1020.929,190.825,-120.623,168.298,50.090,159.395
C06285=1020.923,190.576,-120.600,168.295,50.096,159.396
C06286=1020.918,190.327,-120.576,168.290,50.103,159.396
C06287=1020.913,190.078,-120.553,168.287,50.109,159.397
C06288=1020.908,189.829,-120.531,168.282,50.116,159.398
C06289=1020.903,189.580,-120.508,168.278,50.122,159.398
C06290=1020.897,189.331,-120.485,168.274,50.129,159.399
C06291=1020.892,189.083,-120.462,168.270,50.136,159.400
C06292=1020.887,188.834,-120.439,168.267,50.143,159.401
C06293=1020.881,188.585,-120.416,168.262,50.149,159.401
C06294=1020.876,188.336,-120.394,168.258,50.156,159.402
C06295=1020.871,188.087,-120.370,168.254,50.163,159.403
C06296=1020.864,187.805,-120.345,168.249,50.170,159.403
C06297=1020.859,187.524,-120.319,168.245,50.178,159.404
C06298=1020.853,187.242,-120.293,168.241,50.185,159.405
C06299=1020.847,186.961,-120.267,168.235,50.193,159.406
C06300=1020.842,186.713,-120.244,168.232,50.199,159.406
C06301=1020.837,186.463,-120.222,168.228,50.206,159.407
C06302=1020.832,186.214,-120.199,168.224,50.212,159.408
C06303=1020.826,185.966,-120.176,168.220,50.219,159.409
C06304=1020.821,185.716,-120.153,168.217,50.226,159.409
C06305=1020.817,185.468,-120.131,168.212,50.232,159.410
C06306=1020.811,185.219,-120.108,168.208,50.239,159.411
C06307=1020.806,184.969,-120.084,168.204,50.246,159.411
C06308=1020.801,184.721,-120.062,168.200,50.253,159.412
C06309=1020.795,184.472,-120.039,168.196,50.259,159.413
C06310=1020.791,184.223,-120.016,168.192,50.266,159.413
C06311=1020.785,183.974,-119.994,168.188,50.273,159.414
C06312=1020.780,183.726,-119.971,168.184,50.279,159.415
C06313=1020.775,183.476,-119.949,168.180,50.286,159.415
C06314=1020.771,183.228,-119.926,168.177,50.292,159.416
C06315=1020.765,182.979,-119.903,168.173,50.299,159.417
C06316=1020.759,182.729,-119.881,168.169,50.305,159.418
C06317=1020.755,182.481,-119.858,168.165,50.312,159.418
C06318=1020.750,182.231,-119.835,168.161,50.319,159.419
C06319=1020.744,181.982,-119.812,168.158,50.326,159.420
C06320=1020.739,181.733,-119.791,168.153,50.333,159.421
C06321=1020.733,181.484,-119.769,168.150,50.339,159.421
C06322=1020.728,181.235,-119.747,168.145,50.347,159.422
C06323=1020.722,180.986,-119.724,168.142,50.353,159.423
C06324=1020.717,180.738,-119.703,168.137,50.360,159.424
C06325=1020.711,180.488,-119.681,168.134,50.367,159.424
C06326=1020.706,180.239,-119.658,168.129,50.374,159.425
C06327=1020.700,179.991,-119.636,168.126,50.381,159.426
C06328=1020.695,179.741,-119.614,168.122,50.388,159.427
C06329=1020.690,179.493,-119.592,168.118,50.395,159.427
C06330=1020.684,179.243,-119.571,168.115,50.401,159.428
C06331=1020.679,178.995,-119.549,168.110,50.409,159.429
C06332=1020.673,178.745,-119.527,168.107,50.415,159.430
C06333=1020.667,178.497,-119.505,168.103,50.422,159.430
C06334=1020.662,178.248,-119.482,168.099,50.429,159.431
C06335=1020.657,177.999,-119.461,168.095,50.436,159.432
C06336=1020.652,177.749,-119.438,168.091,50.444,159.433
C06337=1020.646,177.501,-119.417,168.088,50.450,159.434
C06338=1020.641,177.251,-119.395,168.084,50.457,159.434
C06339=1020.636,177.003,-119.373,168.080,50.464,159.435
C06340=1020.630,176.754,-119.351,168.076,50.471,159.436
C06341=1020.625,176.505,-119.329,168.073,50.478,159.437
C06342=1020.619,176.256,-119.307,168.068,50.485,159.437
C06343=1020.614,176.007,-119.285,168.065,50.492,159.438
C06344=1020.608,175.758,-119.263,168.060,50.499,159.439
C06345=1020.603,175.509,-119.242,168.057,50.506,159.440
C06346=1020.598,175.260,-119.220,168.054,50.512,159.440
C06347=1020.592,175.011,-119.198,168.049,50.519,159.441
C06348=1020.587,174.762,-119.176,168.046,50.526,159.442
C06349=1020.581,174.513,-119.154,168.042,50.533,159.443
C06350=1020.577,174.264,-119.132,168.038,50.540,159.443
C06351=1020.571,174.015,-119.111,168.034,50.547,159.444
C06352=1020.566,173.766,-119.089,168.031,50.554,159.445
C06353=1020.561,173.517,-119.067,168.027,50.560,159.446
C06354=1020.555,173.268,-119.045,168.023,50.567,159.446
C06355=1020.550,173.019,-119.023,168.019,50.574,159.447
C06356=1020.545,172.770,-119.002,168.016,50.581,159.448
C06357=1020.539,172.521,-118.980,168.012,50.589,159.449
C06358=1020.534,172.272,-118.958,168.009,50.596,159.450
C06359=1020.529,172.023,-118.936,168.005,50.602,159.450
C06360=1020.523,171.741,-118.912,168.001,50.610,159.451
C06361=1020.517,171.459,-118.887,167.997,50.618,159.452
C06362=1020.511,171.177,-118.863,167.992,50.626,159.453
C06363=1020.505,170.896,-118.838,167.988,50.634,159.454
C06364=1020.499,170.646,-118.816,167.984,50.641,159.455
C06365=1020.494,170.398,-118.794,167.981,50.647,159.455
C06366=1020.490,170.149,-118.772,167.978,50.654,159.456
C06367=1020.484,169.899,-118.752,167.973,50.661,159.457
C06368=1020.479,169.650,-118.730,167.970,50.668,159.458
C06369=1020.473,169.402,-118.708,167.966,50.675,159.458
C06370=1020.468,169.152,-118.686,167.963,50.682,159.459
C06371=1020.463,168.903,-118.664,167.958,50.689,159.460
C06372=1020.458,168.655,-118.643,167.955,50.696,159.461
C06373=1020.453,168.405,-118.622,167.952,50.703,159.461
C06374=1020.448,168.156,-118.600,167.948,50.709,159.462
C06375=1020.442,167.907,-118.578,167.945,50.716,159.463
C06376=1020.437,167.659,-118.557,167.940,50.723,159.464
C06377=1020.432,167.410,-118.535,167.937,50.730,159.464
C06378=1020.427,167.160,-118.514,167.933,50.737,159.465
C06379=1020.422,166.911,-118.492,167.930,50.744,159.466
C06380=1020.416,166.663,-118.471,167.927,50.750,159.467
C06381=1020.411,166.414,-118.449,167.923,50.757,159.468
C06382=1020.406,166.164,-118.427,167.919,50.764,159.468
C06383=1020.401,165.915,-118.406,167.915,50.771,159.469
C06384=1020.396,165.666,-118.384,167.912,50.778,159.470
C06385=1020.391,165.417,-118.363,167.909,50.785,159.471
C06386=1020.386,165.168,-118.342,167.905,50.792,159.471
C06387=1020.380,164.919,-118.319,167.902,50.798,159.472
C06388=1020.375,164.670,-118.298,167.897,50.806,159.473
C06389=1020.370,164.421,-118.277,167.894,50.812,159.474
C06390=1020.365,164.172,-118.255,167.891,50.819,159.474
C06391=1020.360,163.924,-118.234,167.887,50.826,159.475
C06392=1020.355,163.674,-118.213,167.884,50.833,159.476
C06393=1020.350,163.425,-118.191,167.880,50.840,159.477
C06394=1020.345,163.176,-118.170,167.877,50.847,159.478
C06395=1020.340,162.927,-118.148,167.874,50.853,159.478
C06396=1020.334,162.678,-118.127,167.869,50.861,159.479
C06397=1020.330,162.429,-118.106,167.866,50.867,159.480
C06398=1020.325,162.180,-118.084,167.862,50.874,159.481
C06399=1020.319,161.932,-118.063,167.859,50.881,159.481
C06400=1020.314,161.681,-118.041,167.856,50.888,159.482
C06401=1020.309,161.433,-118.019,167.852,50.895,159.483
C06402=1020.304,161.183,-117.999,167.849,50.902,159.484
C06403=1020.299,160.935,-117.977,167.845,50.908,159.485
C06404=1020.294,160.685,-117.956,167.842,50.915,159.485
C06405=1020.289,160.437,-117.934,167.839,50.922,159.486
C06406=1020.285,160.188,-117.912,167.835,50.929,159.487
C06407=1020.279,159.939,-117.892,167.832,50.936,159.488
C06408=1020.274,159.690,-117.870,167.828,50.943,159.488
C06409=1020.269,159.441,-117.850,167.824,50.950,159.489
C06410=1020.264,159.192,-117.828,167.821,50.957,159.490
C06411=1020.260,158.943,-117.806,167.817,50.963,159.491
C06412=1020.254,158.693,-117.786,167.814,50.970,159.492
C06413=1020.248,158.444,-117.764,167.811,50.978,159.493
C06414=1020.243,158.195,-117.744,167.808,50.985,159.493
C06415=1020.239,157.946,-117.723,167.804,50.991,159.494
C06416=1020.233,157.697,-117.701,167.801,50.998,159.495
C06417=1020.228,157.448,-117.681,167.796,51.005,159.496
C06418=1020.223,157.199,-117.660,167.793,51.013,159.497
C06419=1020.217,156.950,-117.640,167.790,51.020,159.497
C06420=1020.212,156.701,-117.618,167.787,51.027,159.498
C06421=1020.207,156.452,-117.597,167.783,51.034,159.499
C06422=1020.202,156.203,-117.577,167.780,51.041,159.500
C06423=1020.197,155.954,-117.556,167.777,51.048,159.501
C06424=1020.191,155.672,-117.532,167.773,51.056,159.502
C06425=1020.184,155.389,-117.509,167.769,51.064,159.502
C06426=1020.178,155.107,-117.485,167.765,51.072,159.503
C06427=1020.172,154.825,-117.461,167.761,51.080,159.504
C06428=1020.167,154.575,-117.441,167.758,51.087,159.505
C06429=1020.162,154.326,-117.420,167.755,51.094,159.506
C06430=1020.157,154.077,-117.399,167.751,51.101,159.507
C06431=1020.151,153.828,-117.379,167.747,51.108,159.507
C06432=1020.147,153.579,-117.358,167.744,51.115,159.508
C06433=1020.142,153.330,-117.337,167.741,51.122,159.509
C06434=1020.136,153.080,-117.317,167.737,51.129,159.510
C06435=1020.131,152.832,-117.295,167.734,51.136,159.511
C06436=1020.126,152.583,-117.275,167.731,51.143,159.512
C06437=1020.120,152.334,-117.254,167.728,51.151,159.513
C06438=1020.115,152.085,-117.234,167.724,51.157,159.513
C06439=1020.110,151.835,-117.213,167.721,51.164,159.514
C06440=1020.104,151.586,-117.193,167.718,51.171,159.515
C06441=1020.099,151.337,-117.172,167.714,51.179,159.516
C06442=1020.094,151.088,-117.152,167.710,51.186,159.517
C06443=1020.089,150.839,-117.131,167.707,51.193,159.517
C06444=1020.084,150.590,-117.111,167.704,51.200,159.518
C06445=1020.079,150.341,-117.090,167.701,51.207,159.519
C06446=1020.074,150.092,-117.070,167.697,51.214,159.520
C06447=1020.068,149.843,-117.049,167.694,51.221,159.521
C06448=1020.063,149.593,-117.029,167.691,51.228,159.521
C06449=1020.058,149.344,-117.009,167.687,51.235,159.522
C06450=1020.053,149.095,-116.988,167.684,51.242,159.523
C06451=1020.048,148.846,-116.968,167.681,51.249,159.524
C06452=1020.042,148.597,-116.947,167.678,51.256,159.525
C06453=1020.037,148.348,-116.927,167.674,51.263,159.526
C06454=1020.032,148.099,-116.906,167.671,51.271,159.527
C06455=1020.027,147.849,-116.885,167.668,51.278,159.527
C06456=1020.021,147.601,-116.865,167.665,51.285,159.528
C06457=1020.016,147.352,-116.845,167.660,51.292,159.529
C06458=1020.011,147.103,-116.825,167.657,51.299,159.530
C06459=1020.006,146.853,-116.805,167.654,51.306,159.531
C06460=1020.000,146.604,-116.784,167.651,51.313,159.531
C06461=1019.995,146.355,-116.764,167.647,51.320,159.532
C06462=1019.990,146.106,-116.743,167.645,51.328,159.533
C06463=1019.985,145.856,-116.723,167.641,51.335,159.534
C06464=1019.980,145.607,-116.703,167.638,51.341,159.535
C06465=1019.974,145.359,-116.683,167.635,51.349,159.536
C06466=1019.969,145.110,-116.663,167.632,51.356,159.536
C06467=1019.964,144.860,-116.643,167.628,51.363,159.537
C06468=1019.959,144.611,-116.622,167.625,51.370,159.538
C06469=1019.953,144.362,-116.602,167.622,51.377,159.539
C06470=1019.948,144.112,-116.582,167.619,51.384,159.540
C06471=1019.943,143.863,-116.562,167.616,51.392,159.541
C06472=1019.937,143.615,-116.542,167.613,51.399,159.542
C06473=1019.932,143.366,-116.523,167.609,51.406,159.542
C06474=1019.927,143.116,-116.502,167.606,51.413,159.543
C06475=1019.922,142.867,-116.481,167.603,51.420,159.544
C06476=1019.916,142.618,-116.462,167.599,51.427,159.545
C06477=1019.911,142.369,-116.442,167.596,51.435,159.546
C06478=1019.907,142.120,-116.422,167.592,51.442,159.547
C06479=1019.901,141.871,-116.402,167.589,51.449,159.547
C06480=1019.895,141.622,-116.382,167.586,51.456,159.548
C06481=1019.890,141.372,-116.362,167.583,51.463,159.549
C06482=1019.884,141.123,-116.342,167.580,51.470,159.550
C06483=1019.880,140.874,-116.322,167.576,51.477,159.551
C06484=1019.875,140.625,-116.302,167.573,51.485,159.552
C06485=1019.869,140.376,-116.281,167.570,51.492,159.552
C06486=1019.864,140.126,-116.262,167.567,51.499,159.553
C06487=1019.859,139.878,-116.242,167.564,51.506,159.554
C06488=1019.853,139.596,-116.219,167.561,51.514,159.555
C06489=1019.847,139.313,-116.197,167.557,51.522,159.556
C06490=1019.841,139.030,-116.174,167.553,51.530,159.557
C06491=1019.835,138.748,-116.151,167.549,51.538,159.558
C06492=1019.831,138.499,-116.132,167.546,51.546,159.559
C06493=1019.825,138.250,-116.112,167.543,51.552,159.560
C06494=1019.820,138.000,-116.092,167.540,51.559,159.560
C06495=1019.815,137.751,-116.071,167.537,51.567,159.561
C06496=1019.810,137.502,-116.053,167.534,51.574,159.562
C06497=1019.804,137.253,-116.032,167.530,51.581,159.563
C06498=1019.799,137.004,-116.013,167.528,51.589,159.564
C06499=1019.794,136.754,-115.993,167.524,51.596,159.565
C06500=1019.788,136.506,-115.973,167.521,51.602,159.565
C06501=1019.783,136.256,-115.953,167.518,51.610,159.566
C06502=1019.778,136.007,-115.934,167.515,51.617,159.567
C06503=1019.773,135.758,-115.914,167.511,51.624,159.568
C06504=1019.767,135.509,-115.895,167.509,51.632,159.569
C06505=1019.762,135.259,-115.875,167.505,51.639,159.570
C06506=1019.756,135.010,-115.855,167.502,51.646,159.571
C06507=1019.752,134.761,-115.836,167.499,51.653,159.572
C06508=1019.746,134.512,-115.816,167.496,51.660,159.572
C06509=1019.741,134.263,-115.796,167.493,51.668,159.573
C06510=1019.736,134.014,-115.777,167.490,51.675,159.574
C06511=1019.730,133.765,-115.758,167.487,51.682,159.575
C06512=1019.725,133.515,-115.738,167.485,51.689,159.576
C06513=1019.720,133.267,-115.718,167.481,51.696,159.577
C06514=1019.715,133.017,-115.698,167.478,51.703,159.578
C06515=1019.709,132.768,-115.679,167.475,51.711,159.579
C06516=1019.705,132.519,-115.660,167.472,51.718,159.579
C06517=1019.699,132.270,-115.640,167.469,51.724,159.580
C06518=1019.693,132.020,-115.620,167.466,51.732,159.581
C06519=1019.689,131.771,-115.601,167.463,51.739,159.582
C06520=1019.683,131.522,-115.582,167.459,51.746,159.583
C06521=1019.679,131.273,-115.562,167.457,51.754,159.584
C06522=1019.673,131.024,-115.542,167.453,51.761,159.584
C06523=1019.668,130.774,-115.522,167.450,51.768,159.585
C06524=1019.663,130.525,-115.504,167.447,51.775,159.586
C06525=1019.658,130.276,-115.484,167.444,51.782,159.587
C06526=1019.652,130.026,-115.464,167.441,51.789,159.588
C06527=1019.647,129.778,-115.446,167.438,51.797,159.589
C06528=1019.641,129.528,-115.426,167.435,51.804,159.590
C06529=1019.636,129.278,-115.407,167.432,51.812,159.591
C06530=1019.631,129.030,-115.388,167.428,51.819,159.591
C06531=1019.626,128.780,-115.368,167.426,51.826,159.592
C06532=1019.620,128.531,-115.349,167.422,51.833,159.593
C06533=1019.615,128.282,-115.330,167.420,51.841,159.594
C06534=1019.609,128.033,-115.311,167.416,51.848,159.595
C06535=1019.604,127.784,-115.292,167.413,51.855,159.596
C06536=1019.598,127.534,-115.273,167.410,51.863,159.597
C06537=1019.593,127.285,-115.254,167.407,51.870,159.597
C06538=1019.588,127.036,-115.235,167.404,51.877,159.598
C06539=1019.582,126.787,-115.216,167.401,51.884,159.599
C06540=1019.578,126.538,-115.196,167.398,51.892,159.600
C06541=1019.572,126.288,-115.177,167.395,51.899,159.601
C06542=1019.567,126.040,-115.158,167.392,51.907,159.602
C06543=1019.561,125.790,-115.139,167.389,51.914,159.603
C06544=1019.556,125.540,-115.120,167.386,51.921,159.604
C06545=1019.551,125.291,-115.101,167.383,51.928,159.605
C06546=1019.545,125.042,-115.082,167.380,51.936,159.606
C06547=1019.540,124.793,-115.063,167.378,51.943,159.606
C06548=1019.534,124.544,-115.044,167.375,51.950,159.607
C06549=1019.529,124.295,-115.025,167.372,51.957,159.608
C06550=1019.523,124.046,-115.006,167.368,51.964,159.609
C06551=1019.519,123.796,-114.988,167.366,51.972,159.610
C06552=1019.513,123.513,-114.966,167.362,51.980,159.611
C06553=1019.507,123.231,-114.944,167.358,51.988,159.612
C06554=1019.501,122.949,-114.923,167.356,51.996,159.613
C06555=1019.495,122.666,-114.901,167.352,52.005,159.614
C06556=1019.490,122.417,-114.882,167.349,52.012,159.615
C06557=1019.485,122.168,-114.863,167.346,52.019,159.616
C06558=1019.479,121.919,-114.844,167.343,52.026,159.616
C06559=1019.474,121.670,-114.825,167.340,52.034,159.617
C06560=1019.468,121.420,-114.806,167.337,52.041,159.618
C06561=1019.463,121.171,-114.788,167.334,52.049,159.619
C06562=1019.458,120.922,-114.768,167.331,52.056,159.620
C06563=1019.453,120.673,-114.749,167.328,52.062,159.621
C06564=1019.447,120.423,-114.731,167.326,52.070,159.622
C06565=1019.442,120.174,-114.712,167.322,52.077,159.623
C06566=1019.436,119.925,-114.693,167.320,52.085,159.624
C06567=1019.431,119.676,-114.674,167.316,52.092,159.624
C06568=1019.427,119.426,-114.655,167.313,52.099,159.625
C06569=1019.422,119.177,-114.636,167.310,52.107,159.626
C06570=1019.416,118.928,-114.617,167.307,52.114,159.627
C06571=1019.411,118.679,-114.598,167.304,52.121,159.628
C06572=1019.406,118.429,-114.580,167.302,52.128,159.629
C06573=1019.400,118.180,-114.560,167.299,52.135,159.630
C06574=1019.395,117.931,-114.541,167.296,52.142,159.630
C06575=1019.390,117.681,-114.523,167.293,52.150,159.631
C06576=1019.385,117.433,-114.504,167.290,52.157,159.632
C06577=1019.380,117.184,-114.485,167.287,52.164,159.633
C06578=1019.374,116.934,-114.467,167.284,52.171,159.634
C06579=1019.369,116.685,-114.448,167.282,52.178,159.635
C06580=1019.364,116.436,-114.429,167.278,52.185,159.636
C06581=1019.359,116.186,-114.410,167.276,52.193,159.637
C06582=1019.354,115.938,-114.392,167.273,52.200,159.637
C06583=1019.348,115.688,-114.372,167.269,52.207,159.638
C06584=1019.343,115.439,-114.354,167.266,52.214,159.639
C06585=1019.338,115.189,-114.334,167.264,52.221,159.640
C06586=1019.333,114.940,-114.315,167.261,52.228,159.641
C06587=1019.328,114.691,-114.297,167.258,52.235,159.642
C06588=1019.323,114.441,-114.278,167.255,52.243,159.643
C06589=1019.318,114.192,-114.260,167.252,52.250,159.643
C06590=1019.313,113.943,-114.241,167.250,52.257,159.644
C06591=1019.307,113.694,-114.222,167.247,52.264,159.645
C06592=1019.302,113.445,-114.204,167.244,52.272,159.646
C06593=1019.297,113.196,-114.185,167.241,52.279,159.647
C06594=1019.292,112.946,-114.166,167.238,52.286,159.648
C06595=1019.287,112.697,-114.147,167.235,52.293,159.649
C06596=1019.282,112.448,-114.129,167.233,52.300,159.650
C06597=1019.276,112.198,-114.110,167.230,52.307,159.650
C06598=1019.272,111.949,-114.092,167.226,52.314,159.651
C06599=1019.266,111.700,-114.073,167.224,52.322,159.652
C06600=1019.260,111.450,-114.055,167.220,52.329,159.653
C06601=1019.256,111.201,-114.037,167.218,52.337,159.654
C06602=1019.250,110.952,-114.018,167.216,52.344,159.655
C06603=1019.245,110.702,-113.999,167.212,52.351,159.656
C06604=1019.239,110.454,-113.981,167.210,52.358,159.657
C06605=1019.235,110.205,-113.963,167.207,52.366,159.657
C06606=1019.229,109.955,-113.944,167.204,52.373,159.658
C06607=1019.224,109.706,-113.925,167.201,52.380,159.659
C06608=1019.219,109.457,-113.908,167.197,52.387,159.660
C06609=1019.213,109.207,-113.889,167.196,52.395,159.661
C06610=1019.208,108.958,-113.870,167.193,52.402,159.662
C06611=1019.203,108.709,-113.853,167.190,52.410,159.663
C06612=1019.197,108.459,-113.834,167.187,52.417,159.664
C06613=1019.192,108.210,-113.817,167.184,52.424,159.665
C06614=1019.187,107.961,-113.798,167.181,52.432,159.665
C06615=1019.182,107.712,-113.780,167.178,52.439,159.667
C06616=1019.175,107.428,-113.759,167.175,52.447,159.668
C06617=1019.169,107.146,-113.739,167.172,52.456,159.669
C06618=1019.163,106.864,-113.718,167.168,52.464,159.669
C06619=1019.157,106.582,-113.698,167.166,52.472,159.670
C06620=1019.152,106.332,-113.680,167.163,52.480,159.671
C06621=1019.147,106.082,-113.661,167.160,52.487,159.672
C06622=1019.141,105.834,-113.643,167.157,52.494,159.673
C06623=1019.136,105.585,-113.625,167.154,52.502,159.674
C06624=1019.130,105.335,-113.607,167.151,52.509,159.675
C06625=1019.125,105.086,-113.589,167.148,52.516,159.676
C06626=1019.120,104.837,-113.571,167.145,52.523,159.677
C06627=1019.115,104.587,-113.553,167.143,52.531,159.678
C06628=1019.109,104.338,-113.534,167.140,52.538,159.679
C06629=1019.104,104.089,-113.516,167.137,52.546,159.680
C06630=1019.099,103.839,-113.498,167.134,52.553,159.680
C06631=1019.094,103.590,-113.481,167.131,52.560,159.681
C06632=1019.089,103.341,-113.463,167.128,52.568,159.682
C06633=1019.083,103.091,-113.445,167.126,52.574,159.683
C06634=1019.078,102.842,-113.426,167.124,52.582,159.684
C06635=1019.073,102.592,-113.408,167.120,52.589,159.685
C06636=1019.068,102.343,-113.391,167.117,52.596,159.686
C06637=1019.062,102.095,-113.372,167.115,52.604,159.687
C06638=1019.056,101.845,-113.354,167.112,52.611,159.687
C06639=1019.052,101.596,-113.336,167.109,52.618,159.688
C06640=1019.046,101.347,-113.318,167.107,52.626,159.689
C06641=1019.041,101.097,-113.300,167.104,52.633,159.690
C06642=1019.036,100.848,-113.282,167.100,52.640,159.691
C06643=1019.031,100.599,-113.264,167.098,52.648,159.692
C06644=1019.026,100.349,-113.246,167.096,52.655,159.693
C06645=1019.020,100.100,-113.228,167.093,52.662,159.694
C06646=1019.015,99.850,-113.210,167.090,52.669,159.695
C06647=1019.010,99.601,-113.192,167.087,52.677,159.695
C06648=1019.005,99.352,-113.174,167.085,52.683,159.696
C06649=1018.999,99.103,-113.157,167.082,52.691,159.697
C06650=1018.994,98.853,-113.138,167.079,52.698,159.698
C06651=1018.989,98.604,-113.121,167.076,52.706,159.699
C06652=1018.983,98.355,-113.103,167.073,52.713,159.700
C06653=1018.978,98.106,-113.085,167.070,52.721,159.701
C06654=1018.973,97.856,-113.068,167.067,52.728,159.702
C06655=1018.968,97.607,-113.050,167.065,52.736,159.703
C06656=1018.962,97.358,-113.033,167.063,52.743,159.704
C06657=1018.956,97.108,-113.015,167.060,52.750,159.705
C06658=1018.951,96.859,-112.997,167.057,52.758,159.705
C06659=1018.946,96.610,-112.979,167.054,52.765,159.706
C06660=1018.940,96.360,-112.962,167.051,52.773,159.707
C06661=1018.936,96.111,-112.944,167.048,52.780,159.708
C06662=1018.930,95.862,-112.927,167.045,52.787,159.709
C06663=1018.925,95.613,-112.909,167.043,52.794,159.710
C06664=1018.919,95.364,-112.892,167.041,52.802,159.711
C06665=1018.914,95.113,-112.874,167.037,52.809,159.712
C06666=1018.908,94.864,-112.856,167.034,52.816,159.712
C06667=1018.903,94.615,-112.839,167.032,52.824,159.713
C06668=1018.897,94.366,-112.821,167.029,52.831,159.714
C06669=1018.893,94.116,-112.803,167.027,52.839,159.715
C06670=1018.887,93.867,-112.786,167.024,52.846,159.716
C06671=1018.882,93.618,-112.768,167.021,52.853,159.717
C06672=1018.876,93.369,-112.751,167.018,52.861,159.718
C06673=1018.872,93.119,-112.733,167.015,52.868,159.719
C06674=1018.866,92.870,-112.716,167.012,52.876,159.720
C06675=1018.861,92.621,-112.698,167.010,52.883,159.721
C06676=1018.855,92.372,-112.681,167.007,52.890,159.721
C06677=1018.851,92.122,-112.663,167.005,52.898,159.722
C06678=1018.845,91.873,-112.646,167.002,52.905,159.723
C06679=1018.840,91.623,-112.628,166.999,52.912,159.724
C06680=1018.835,91.376,-112.610,166.997,52.919,159.725
C06681=1018.829,91.129,-112.593,166.994,52.926,159.726
C06682=1018.824,90.882,-112.576,166.991,52.934,159.727
C06683=1018.819,90.636,-112.558,166.988,52.941,159.727
C06684=1018.814,90.389,-112.541,166.986,52.948,159.729
C06685=1018.808,90.143,-112.524,166.983,52.955,159.729
C06686=1018.804,89.896,-112.507,166.980,52.962,159.730
C06687=1018.798,89.649,-112.490,166.978,52.969,159.731
C06688=1018.793,89.400,-112.472,166.975,52.977,159.732
C06689=1018.788,89.150,-112.455,166.972,52.984,159.733
C06690=1018.783,88.901,-112.437,166.970,52.992,159.734
C06691=1018.777,88.652,-112.420,166.967,52.999,159.735
C06692=1018.772,88.402,-112.403,166.963,53.006,159.735
C06693=1018.766,88.153,-112.385,166.962,53.014,159.737
C06694=1018.761,87.904,-112.368,166.959,53.021,159.737
C06695=1018.756,87.654,-112.351,166.956,53.029,159.738
C06696=1018.750,87.405,-112.334,166.953,53.036,159.739
C06697=1018.745,87.156,-112.318,166.951,53.044,159.740
C06698=1018.739,86.907,-112.300,166.947,53.051,159.741
C06699=1018.734,86.657,-112.283,166.945,53.059,159.742
C06700=1018.728,86.408,-112.266,166.943,53.066,159.743
C06701=1018.723,86.158,-112.249,166.940,53.074,159.744
C06702=1018.718,85.909,-112.231,166.937,53.081,159.745
C06703=1018.712,85.659,-112.214,166.935,53.089,159.746
C06704=1018.707,85.410,-112.197,166.931,53.096,159.746
C06705=1018.702,85.161,-112.180,166.928,53.103,159.747
C06706=1018.696,84.911,-112.163,166.926,53.111,159.748
C06707=1018.691,84.662,-112.145,166.924,53.118,159.749
C06708=1018.686,84.412,-112.129,166.921,53.126,159.750
C06709=1018.680,84.163,-112.112,166.918,53.133,159.751
C06710=1018.675,83.914,-112.094,166.916,53.141,159.752
C06711=1018.670,83.664,-112.077,166.913,53.148,159.753
C06712=1018.663,83.415,-112.060,166.909,53.155,159.754
C06713=1018.658,83.166,-112.044,166.908,53.162,159.755
C06714=1018.654,82.917,-112.027,166.905,53.170,159.755
C06715=1018.648,82.668,-112.009,166.902,53.177,159.756
C06716=1018.643,82.418,-111.993,166.899,53.185,159.757
C06717=1018.638,82.168,-111.976,166.896,53.192,159.758
C06718=1018.632,81.919,-111.958,166.895,53.199,159.759
C06719=1018.627,81.670,-111.941,166.892,53.207,159.760
C06720=1018.622,81.420,-111.925,166.889,53.214,159.761
C06721=1018.616,81.171,-111.907,166.886,53.222,159.762
C06722=1018.611,80.921,-111.890,166.883,53.229,159.763
C06723=1018.606,80.672,-111.873,166.881,53.236,159.764
C06724=1018.601,80.423,-111.856,166.878,53.244,159.765
C06725=1018.596,80.174,-111.839,166.875,53.251,159.765
C06726=1018.590,79.924,-111.822,166.872,53.258,159.766
C06727=1018.584,79.675,-111.805,166.870,53.266,159.767
C06728=1018.579,79.426,-111.789,166.868,53.273,159.768
C06729=1018.574,79.176,-111.772,166.865,53.280,159.769
C06730=1018.569,78.926,-111.755,166.862,53.288,159.770
C06731=1018.564,78.678,-111.738,166.859,53.295,159.771
C06732=1018.557,78.390,-111.718,166.857,53.303,159.772
C06733=1018.552,78.102,-111.699,166.854,53.312,159.773
C06734=1018.545,77.815,-111.679,166.850,53.320,159.774
C06735=1018.540,77.527,-111.660,166.848,53.329,159.775
C06736=1018.534,77.277,-111.643,166.845,53.336,159.776
C06737=1018.529,77.028,-111.626,166.842,53.343,159.776
C06738=1018.523,76.779,-111.609,166.839,53.351,159.777
C06739=1018.518,76.529,-111.592,166.836,53.358,159.778
C06740=1018.513,76.280,-111.575,166.834,53.365,159.779
C06741=1018.507,76.030,-111.558,166.832,53.373,159.780
C06742=1018.502,75.781,-111.543,166.829,53.380,159.781
C06743=1018.497,75.532,-111.526,166.826,53.388,159.782
C06744=1018.491,75.249,-111.507,166.824,53.396,159.783
C06745=1018.485,74.967,-111.488,166.820,53.404,159.784
C06746=1018.478,74.685,-111.469,166.817,53.413,159.785
C06747=1018.472,74.403,-111.450,166.814,53.421,159.786
C06748=1018.467,74.153,-111.434,166.812,53.429,159.787
C06749=1018.461,73.904,-111.417,166.809,53.436,159.788
C06750=1018.456,73.655,-111.401,166.806,53.443,159.789
C06751=1018.451,73.405,-111.384,166.803,53.451,159.790
C06752=1018.445,73.156,-111.368,166.801,53.458,159.791
C06753=1018.440,72.906,-111.351,166.798,53.465,159.791
C06754=1018.435,72.656,-111.334,166.796,53.473,159.792
C06755=1018.429,72.408,-111.318,166.793,53.481,159.793
C06756=1018.424,72.158,-111.301,166.790,53.489,159.794
C06757=1018.419,71.909,-111.284,166.787,53.496,159.795
C06758=1018.413,71.659,-111.268,166.785,53.503,159.796
C06759=1018.408,71.410,-111.252,166.783,53.511,159.797
C06760=1018.402,71.161,-111.235,166.780,53.518,159.798
C06761=1018.397,70.911,-111.219,166.777,53.525,159.798
C06762=1018.392,70.662,-111.202,166.774,53.533,159.799
C06763=1018.387,70.413,-111.186,166.772,53.540,159.800
C06764=1018.381,70.163,-111.169,166.769,53.547,159.801
C06765=1018.376,69.913,-111.153,166.767,53.555,159.802
C06766=1018.371,69.664,-111.137,166.764,53.562,159.803
C06767=1018.366,69.415,-111.120,166.761,53.569,159.804
C06768=1018.360,69.165,-111.104,166.759,53.577,159.805
C06769=1018.355,68.916,-111.087,166.756,53.584,159.806
C06770=1018.349,68.667,-111.071,166.754,53.591,159.807
C06771=1018.344,68.417,-111.054,166.751,53.599,159.807
C06772=1018.339,68.168,-111.037,166.748,53.607,159.808
C06773=1018.333,67.918,-111.022,166.746,53.613,159.809
C06774=1018.328,67.669,-111.006,166.744,53.621,159.810
C06775=1018.323,67.419,-110.989,166.741,53.629,159.811
C06776=1018.317,67.170,-110.973,166.738,53.636,159.812
C06777=1018.312,66.921,-110.956,166.735,53.644,159.813
C06778=1018.307,66.671,-110.941,166.732,53.651,159.814
C06779=1018.301,66.421,-110.924,166.730,53.658,159.815
C06780=1018.296,66.173,-110.908,166.728,53.666,159.816
C06781=1018.291,65.923,-110.891,166.725,53.673,159.816
C06782=1018.285,65.673,-110.876,166.722,53.680,159.817
C06783=1018.279,65.424,-110.859,166.719,53.688,159.818
C06784=1018.275,65.175,-110.843,166.716,53.696,159.819
C06785=1018.269,64.926,-110.827,166.714,53.702,159.820
C06786=1018.264,64.675,-110.811,166.712,53.710,159.821
C06787=1018.258,64.427,-110.795,166.709,53.718,159.822
C06788=1018.253,64.177,-110.778,166.707,53.726,159.823
C06789=1018.248,63.927,-110.762,166.704,53.733,159.824
C06790=1018.242,63.678,-110.746,166.701,53.740,159.824
C06791=1018.237,63.429,-110.730,166.699,53.748,159.826
C06792=1018.231,63.179,-110.714,166.696,53.755,159.826
C06793=1018.226,62.930,-110.698,166.693,53.762,159.827
C06794=1018.221,62.680,-110.682,166.691,53.770,159.828
C06795=1018.215,62.430,-110.666,166.688,53.777,159.829
C06796=1018.210,62.181,-110.651,166.685,53.785,159.830
C06797=1018.204,61.932,-110.634,166.682,53.793,159.831
C06798=1018.199,61.682,-110.619,166.680,53.801,159.832
C06799=1018.193,61.433,-110.603,166.677,53.808,159.833
C06800=1018.188,61.183,-110.587,166.675,53.816,159.834
C06801=1018.182,60.935,-110.571,166.673,53.823,159.834
C06802=1018.177,60.685,-110.556,166.670,53.831,159.836
C06803=1018.171,60.435,-110.540,166.667,53.838,159.836
C06804=1018.166,60.186,-110.525,166.664,53.845,159.837
C06805=1018.160,59.936,-110.508,166.662,53.853,159.838
C06806=1018.155,59.687,-110.492,166.659,53.861,159.839
C06807=1018.149,59.438,-110.476,166.657,53.869,159.840
C06808=1018.143,59.155,-110.459,166.653,53.877,159.841
C06809=1018.137,58.873,-110.441,166.651,53.886,159.842
C06810=1018.130,58.590,-110.423,166.648,53.894,159.843
C06811=1018.124,58.308,-110.405,166.644,53.902,159.844
C06812=1018.119,58.059,-110.390,166.642,53.910,159.845
C06813=1018.114,57.809,-110.374,166.640,53.917,159.846
C06814=1018.108,57.560,-110.358,166.637,53.925,159.847
C06815=1018.103,57.310,-110.343,166.634,53.933,159.848
C06816=1018.097,57.061,-110.326,166.632,53.941,159.849
C06817=1018.092,56.812,-110.311,166.629,53.948,159.849
C06818=1018.086,56.562,-110.296,166.626,53.955,159.850
C06819=1018.081,56.313,-110.280,166.624,53.963,159.851
C06820=1018.075,56.063,-110.264,166.621,53.970,159.852
C06821=1018.070,55.814,-110.249,166.618,53.978,159.853
C06822=1018.064,55.564,-110.233,166.616,53.985,159.854
C06823=1018.059,55.315,-110.217,166.614,53.993,159.855
C06824=1018.054,55.065,-110.202,166.611,54.000,159.856
C06825=1018.048,54.816,-110.186,166.608,54.008,159.857
C06826=1018.043,54.567,-110.171,166.605,54.015,159.857
C06827=1018.038,54.316,-110.154,166.602,54.022,159.858
C06828=1018.032,54.068,-110.138,166.600,54.030,159.859
C06829=1018.027,53.818,-110.123,166.598,54.037,159.860
C06830=1018.022,53.568,-110.108,166.595,54.045,159.861
C06831=1018.016,53.319,-110.092,166.593,54.053,159.862
C06832=1018.011,53.070,-110.076,166.590,54.060,159.863
C06833=1018.005,52.820,-110.061,166.587,54.067,159.864
C06834=1018.000,52.571,-110.045,166.585,54.075,159.865
C06835=1017.994,52.321,-110.029,166.582,54.083,159.865
C06836=1017.989,52.072,-110.014,166.580,54.090,159.866
C06837=1017.983,51.822,-109.999,166.577,54.097,159.867
C06838=1017.978,51.573,-109.983,166.575,54.105,159.868
C06839=1017.972,51.323,-109.967,166.572,54.112,159.869
C06840=1017.967,51.074,-109.952,166.569,54.119,159.870
C06841=1017.962,50.825,-109.937,166.566,54.127,159.871
C06842=1017.956,50.576,-109.921,166.564,54.134,159.872
C06843=1017.952,50.326,-109.905,166.562,54.142,159.873
C06844=1017.946,50.076,-109.889,166.559,54.149,159.873
C06845=1017.941,49.827,-109.874,166.556,54.156,159.874
C06846=1017.935,49.577,-109.858,166.553,54.164,159.875
C06847=1017.930,49.328,-109.843,166.552,54.171,159.876
C06848=1017.925,49.078,-109.827,166.549,54.179,159.877
C06849=1017.920,48.829,-109.812,166.546,54.186,159.878
C06850=1017.915,48.580,-109.797,166.543,54.194,159.879
C06851=1017.909,48.330,-109.781,166.541,54.201,159.879
C06852=1017.904,48.081,-109.765,166.539,54.208,159.880
C06853=1017.898,47.831,-109.750,166.536,54.216,159.881
C06854=1017.893,47.582,-109.735,166.533,54.223,159.882
C06855=1017.888,47.333,-109.720,166.530,54.230,159.883
C06856=1017.882,47.083,-109.704,166.528,54.238,159.884
C06857=1017.877,46.834,-109.688,166.526,54.245,159.885
C06858=1017.871,46.584,-109.673,166.523,54.252,159.886
C06859=1017.866,46.335,-109.657,166.520,54.260,159.886
C06860=1017.861,46.085,-109.642,166.517,54.267,159.887
C06861=1017.856,45.835,-109.627,166.514,54.274,159.888
C06862=1017.851,45.586,-109.611,166.513,54.281,159.889
C06863=1017.846,45.337,-109.596,166.510,54.289,159.890
C06864=1017.841,45.087,-109.580,166.507,54.297,159.891
C06865=1017.835,44.838,-109.564,166.504,54.304,159.892
C06866=1017.830,44.588,-109.549,166.503,54.311,159.892
C06867=1017.825,44.339,-109.534,166.500,54.318,159.893
C06868=1017.820,44.089,-109.518,166.497,54.326,159.894
C06869=1017.814,43.839,-109.503,166.494,54.333,159.895
C06870=1017.809,43.590,-109.488,166.492,54.340,159.896
C06871=1017.804,43.341,-109.472,166.489,54.347,159.897
C06872=1017.798,43.059,-109.455,166.486,54.356,159.897
C06873=1017.792,42.776,-109.438,166.484,54.364,159.898
C06874=1017.786,42.494,-109.421,166.480,54.372,159.899
C06875=1017.780,42.211,-109.403,166.478,54.380,159.900
C06876=1017.775,41.962,-109.388,166.475,54.388,159.901
C06877=1017.769,41.712,-109.373,166.473,54.396,159.902
C06878=1017.764,41.463,-109.357,166.470,54.403,159.903
C06879=1017.758,41.214,-109.343,166.467,54.410,159.904
C06880=1017.752,40.964,-109.327,166.464,54.418,159.905
C06881=1017.748,40.714,-109.313,166.463,54.425,159.906
C06882=1017.743,40.465,-109.298,166.460,54.433,159.907
C06883=1017.736,40.215,-109.283,166.457,54.440,159.907
C06884=1017.731,39.966,-109.268,166.454,54.447,159.908
C06885=1017.726,39.716,-109.252,166.452,54.455,159.909
C06886=1017.721,39.466,-109.237,166.449,54.463,159.910
C06887=1017.715,39.217,-109.222,166.446,54.470,159.911
C06888=1017.710,38.968,-109.208,166.445,54.477,159.912
C06889=1017.705,38.718,-109.193,166.442,54.485,159.913
C06890=1017.699,38.468,-109.177,166.439,54.492,159.913
C06891=1017.694,38.219,-109.162,166.436,54.499,159.914
C06892=1017.688,37.970,-109.147,166.434,54.507,159.915
C06893=1017.683,37.721,-109.132,166.431,54.515,159.916
C06894=1017.678,37.470,-109.117,166.429,54.522,159.917
C06895=1017.672,37.221,-109.103,166.426,54.529,159.918
C06896=1017.667,36.972,-109.088,166.423,54.536,159.919
C06897=1017.662,36.722,-109.072,166.421,54.544,159.919
C06898=1017.657,36.472,-109.058,166.418,54.551,159.920
C06899=1017.651,36.223,-109.043,166.416,54.559,159.921
C06900=1017.646,35.974,-109.028,166.414,54.566,159.922
C06901=1017.640,35.724,-109.014,166.411,54.574,159.923
C06902=1017.635,35.474,-108.998,166.408,54.581,159.924
C06903=1017.629,35.225,-108.984,166.406,54.589,159.925
C06904=1017.624,34.976,-108.969,166.403,54.596,159.926
C06905=1017.618,34.726,-108.954,166.400,54.604,159.926
C06906=1017.613,34.476,-108.940,166.397,54.611,159.927
C06907=1017.608,34.227,-108.925,166.395,54.619,159.928
C06908=1017.602,33.978,-108.910,166.392,54.627,159.929
C06909=1017.597,33.728,-108.896,166.389,54.634,159.930
C06910=1017.591,33.478,-108.881,166.388,54.641,159.931
C06911=1017.586,33.229,-108.867,166.385,54.648,159.932
C06912=1017.581,32.979,-108.852,166.383,54.656,159.933
C06913=1017.575,32.730,-108.837,166.380,54.664,159.933
C06914=1017.570,32.481,-108.823,166.377,54.671,159.934
C06915=1017.564,32.231,-108.808,166.374,54.679,159.935
C06916=1017.559,31.981,-108.793,166.371,54.686,159.936
C06917=1017.553,31.732,-108.779,166.369,54.693,159.937
C06918=1017.549,31.482,-108.764,166.366,54.701,159.938
C06919=1017.543,31.233,-108.750,166.364,54.708,159.939
C06920=1017.538,30.983,-108.735,166.362,54.716,159.939
C06921=1017.532,30.734,-108.720,166.359,54.723,159.940
C06922=1017.527,30.484,-108.706,166.356,54.731,159.941
C06923=1017.521,30.235,-108.691,166.353,54.738,159.942
C06924=1017.517,29.985,-108.677,166.351,54.745,159.943
C06925=1017.511,29.736,-108.662,166.348,54.753,159.943
C06926=1017.506,29.486,-108.648,166.347,54.761,159.945
C06927=1017.500,29.237,-108.633,166.344,54.768,159.945
C06928=1017.495,28.987,-108.618,166.341,54.775,159.946
C06929=1017.489,28.738,-108.604,166.338,54.783,159.947
C06930=1017.484,28.488,-108.589,166.335,54.790,159.948
C06931=1017.479,28.239,-108.575,166.333,54.798,159.949
C06932=1017.474,27.989,-108.560,166.330,54.805,159.949
C06933=1017.468,27.740,-108.546,166.328,54.812,159.950
C06934=1017.463,27.490,-108.531,166.325,54.819,159.951
C06935=1017.458,27.240,-108.517,166.323,54.827,159.952
C06936=1017.451,26.958,-108.501,166.319,54.835,159.953
C06937=1017.445,26.675,-108.484,166.316,54.844,159.954
C06938=1017.439,26.393,-108.468,166.314,54.853,159.955
C06939=1017.433,26.111,-108.452,166.311,54.861,159.956
C06940=1017.427,25.862,-108.438,166.308,54.869,159.957
C06941=1017.422,25.612,-108.423,166.305,54.876,159.957
C06942=1017.417,25.363,-108.409,166.303,54.883,159.958
C06943=1017.411,25.113,-108.395,166.300,54.891,159.959
C06944=1017.406,24.864,-108.381,166.299,54.898,159.960
C06945=1017.401,24.614,-108.367,166.296,54.906,159.961
C06946=1017.395,24.365,-108.352,166.293,54.913,159.962
C06947=1017.390,24.115,-108.338,166.290,54.921,159.963
C06948=1017.384,23.865,-108.324,166.287,54.928,159.963
C06949=1017.379,23.615,-108.310,166.285,54.936,159.964
C06950=1017.373,23.366,-108.295,166.282,54.943,159.965
C06951=1017.368,23.116,-108.281,166.279,54.950,159.966
C06952=1017.362,22.867,-108.267,166.277,54.959,159.967
C06953=1017.357,22.617,-108.253,166.274,54.966,159.968
C06954=1017.352,22.368,-108.238,166.271,54.973,159.968
C06955=1017.346,22.118,-108.224,166.269,54.981,159.969
C06956=1017.341,21.869,-108.210,166.267,54.988,159.970
C06957=1017.336,21.619,-108.196,166.264,54.995,159.971
C06958=1017.330,21.369,-108.182,166.262,55.003,159.972
C06959=1017.325,21.120,-108.168,166.259,55.010,159.973
C06960=1017.319,20.871,-108.154,166.256,55.018,159.973
C06961=1017.314,20.621,-108.140,166.253,55.025,159.974
C06962=1017.309,20.371,-108.125,166.251,55.032,159.975
C06963=1017.304,20.122,-108.112,166.248,55.040,159.976
C06964=1017.298,19.872,-108.098,166.246,55.047,159.977
C06965=1017.293,19.623,-108.084,166.243,55.054,159.978
C06966=1017.288,19.373,-108.069,166.241,55.062,159.978
C06967=1017.282,19.124,-108.055,166.238,55.069,159.979
C06968=1017.277,18.874,-108.041,166.235,55.077,159.980
C06969=1017.271,18.625,-108.027,166.233,55.085,159.981
C06970=1017.266,18.375,-108.013,166.230,55.092,159.982
C06971=1017.260,18.126,-107.999,166.227,55.100,159.983
C06972=1017.255,17.876,-107.985,166.225,55.107,159.983
C06973=1017.249,17.626,-107.972,166.222,55.114,159.984
C06974=1017.244,17.376,-107.957,166.219,55.122,159.985
C06975=1017.239,17.127,-107.943,166.217,55.129,159.986
C06976=1017.234,16.878,-107.930,166.215,55.136,159.987
C06977=1017.229,16.628,-107.916,166.212,55.144,159.988
C06978=1017.223,16.379,-107.902,166.209,55.151,159.988
C06979=1017.218,16.129,-107.888,166.207,55.159,159.989
C06980=1017.212,15.880,-107.874,166.204,55.166,159.990
C06981=1017.207,15.630,-107.860,166.201,55.174,159.991
C06982=1017.201,15.381,-107.847,166.199,55.181,159.992
C06983=1017.196,15.131,-107.833,166.196,55.189,159.992
C06984=1017.190,14.881,-107.819,166.193,55.196,159.993
C06985=1017.185,14.632,-107.805,166.190,55.203,159.994
C06986=1017.179,14.382,-107.791,166.189,55.211,159.995
C06987=1017.175,14.132,-107.777,166.186,55.218,159.996
C06988=1017.169,13.883,-107.763,166.183,55.225,159.997
C06989=1017.164,13.634,-107.749,166.181,55.233,159.997
C06990=1017.159,13.384,-107.736,166.178,55.240,159.998
C06991=1017.154,13.134,-107.722,166.175,55.248,159.999
C06992=1017.148,12.885,-107.708,166.172,55.255,160.000
C06993=1017.142,12.635,-107.695,166.170,55.263,160.001
C06994=1017.136,12.386,-107.681,166.168,55.271,160.002
C06995=1017.131,12.136,-107.668,166.165,55.278,160.002
C06996=1017.126,11.886,-107.654,166.162,55.286,160.003
C06997=1017.120,11.636,-107.640,166.159,55.293,160.004
C06998=1017.115,11.388,-107.627,166.157,55.301,160.005
C06999=1017.110,11.138,-107.614,166.154,55.308,160.006
C07000=1017.103,10.857,-107.599,166.151,55.317,160.007
C07001=1017.097,10.575,-107.583,166.148,55.325,160.007
C07002=1017.091,10.295,-107.568,166.145,55.334,160.009
C07003=1017.085,10.014,-107.553,166.142,55.342,160.009
C07004=1017.080,9.764,-107.539,166.140,55.350,160.010
C07005=1017.073,9.515,-107.526,166.137,55.357,160.011
C07006=1017.068,9.265,-107.513,166.134,55.365,160.012
C07007=1017.063,9.016,-107.500,166.132,55.373,160.013
C07008=1017.058,8.766,-107.486,166.129,55.380,160.014
C07009=1017.053,8.516,-107.473,166.127,55.388,160.015
C07010=1017.046,8.267,-107.459,166.124,55.395,160.015
C07011=1017.041,8.017,-107.445,166.121,55.403,160.016
C07012=1017.036,7.768,-107.433,166.119,55.410,160.017
C07013=1017.031,7.518,-107.419,166.116,55.418,160.018
C07014=1017.025,7.269,-107.405,166.113,55.425,160.019
C07015=1017.020,7.019,-107.392,166.111,55.433,160.019
C07016=1017.014,6.769,-107.378,166.108,55.440,160.020
C07017=1017.009,6.520,-107.366,166.105,55.448,160.021
C07018=1017.004,6.270,-107.352,166.102,55.455,160.022
C07019=1016.998,6.021,-107.339,166.101,55.462,160.023
C07020=1016.993,5.771,-107.325,166.098,55.470,160.024
C07021=1016.988,5.522,-107.312,166.096,55.477,160.024
C07022=1016.983,5.272,-107.299,166.093,55.485,160.025
C07023=1016.976,5.022,-107.285,166.090,55.491,160.026
C07024=1016.971,4.773,-107.272,166.087,55.499,160.026
C07025=1016.966,4.523,-107.259,166.084,55.506,160.027
C07026=1016.961,4.274,-107.245,166.082,55.514,160.028
C07027=1016.956,4.023,-107.232,166.079,55.521,160.029
C07028=1016.949,3.774,-107.219,166.076,55.529,160.030
C07029=1016.945,3.525,-107.206,166.074,55.536,160.031
C07030=1016.939,3.275,-107.192,166.071,55.544,160.031
C07031=1016.934,3.025,-107.179,166.068,55.551,160.032
C07032=1016.929,2.776,-107.166,166.066,55.559,160.033
C07033=1016.923,2.526,-107.153,166.063,55.566,160.033
C07034=1016.918,2.277,-107.139,166.061,55.573,160.034
C07035=1016.913,2.026,-107.126,166.058,55.580,160.035
C07036=1016.907,1.778,-107.113,166.056,55.588,160.036
C07037=1016.902,1.528,-107.100,166.053,55.595,160.037
C07038=1016.897,1.278,-107.086,166.050,55.603,160.038
C07039=1016.892,1.029,-107.073,166.048,55.610,160.038
C07040=1016.886,0.779,-107.060,166.044,55.617,160.039
C07041=1016.881,0.529,-107.047,166.042,55.625,160.040
C07042=1016.876,0.280,-107.033,166.039,55.632,160.041
C07043=1016.871,0.030,-107.020,166.037,55.640,160.041
C07044=1016.865,-0.220,-107.006,166.035,55.647,160.042
C07045=1016.860,-0.469,-106.994,166.032,55.653,160.043
C07046=1016.854,-0.718,-106.980,166.029,55.661,160.044
C07047=1016.850,-0.968,-106.967,166.027,55.668,160.045
C07048=1016.845,-1.218,-106.954,166.024,55.676,160.045
C07049=1016.838,-1.467,-106.941,166.021,55.683,160.046
C07050=1016.834,-1.717,-106.928,166.018,55.690,160.047
C07051=1016.828,-1.966,-106.914,166.015,55.698,160.048
C07052=1016.823,-2.216,-106.901,166.014,55.705,160.049
C07053=1016.818,-2.466,-106.889,166.011,55.712,160.049
C07054=1016.812,-2.715,-106.875,166.008,55.719,160.050
C07055=1016.808,-2.965,-106.862,166.005,55.727,160.051
C07056=1016.802,-3.214,-106.848,166.002,55.734,160.051
C07057=1016.796,-3.464,-106.836,166.000,55.741,160.052
C07058=1016.792,-3.714,-106.823,165.997,55.749,160.053
C07059=1016.786,-3.963,-106.809,165.995,55.756,160.054
C07060=1016.782,-4.213,-106.796,165.992,55.762,160.054
C07061=1016.776,-4.463,-106.784,165.990,55.770,160.055
C07062=1016.771,-4.713,-106.771,165.987,55.778,160.056
C07063=1016.765,-4.961,-106.758,165.984,55.785,160.057
C07064=1016.759,-5.241,-106.743,165.981,55.794,160.058
C07065=1016.753,-5.519,-106.729,165.978,55.802,160.058
C07066=1016.747,-5.798,-106.715,165.976,55.810,160.059
C07067=1016.740,-6.077,-106.701,165.972,55.819,160.060
C07068=1016.736,-6.327,-106.688,165.970,55.826,160.061
C07069=1016.730,-6.577,-106.675,165.967,55.833,160.062
C07070=1016.725,-6.826,-106.663,165.964,55.840,160.062
C07071=1016.719,-7.076,-106.650,165.961,55.848,160.063
C07072=1016.714,-7.326,-106.638,165.959,55.856,160.064
C07073=1016.709,-7.576,-106.625,165.956,55.863,160.065
C07074=1016.703,-7.825,-106.612,165.954,55.871,160.066
C07075=1016.698,-8.075,-106.600,165.951,55.878,160.066
C07076=1016.693,-8.325,-106.587,165.948,55.885,160.067
C07077=1016.687,-8.574,-106.575,165.945,55.893,160.068
C07078=1016.682,-8.824,-106.561,165.943,55.900,160.069
C07079=1016.676,-9.073,-106.549,165.940,55.908,160.069
C07080=1016.671,-9.323,-106.536,165.937,55.915,160.070
C07081=1016.666,-9.572,-106.523,165.934,55.922,160.071
C07082=1016.660,-9.822,-106.511,165.932,55.930,160.072
C07083=1016.655,-10.071,-106.499,165.929,55.937,160.072
C07084=1016.650,-10.321,-106.485,165.927,55.945,160.073
C07085=1016.644,-10.571,-106.473,165.924,55.952,160.074
C07086=1016.639,-10.821,-106.460,165.921,55.959,160.075
C07087=1016.634,-11.070,-106.448,165.918,55.967,160.075
C07088=1016.629,-11.319,-106.436,165.916,55.974,160.076
C07089=1016.623,-11.569,-106.423,165.913,55.982,160.077
C07090=1016.618,-11.819,-106.410,165.911,55.988,160.078
C07091=1016.612,-12.068,-106.398,165.908,55.996,160.079
C07092=1016.608,-12.318,-106.385,165.906,56.003,160.079
C07093=1016.602,-12.568,-106.373,165.903,56.010,160.080
C07094=1016.597,-12.817,-106.360,165.900,56.018,160.081
C07095=1016.591,-13.067,-106.347,165.898,56.025,160.082
C07096=1016.586,-13.317,-106.336,165.894,56.032,160.082
C07097=1016.582,-13.566,-106.323,165.892,56.040,160.083
C07098=1016.576,-13.816,-106.310,165.889,56.047,160.084
C07099=1016.570,-14.066,-106.298,165.886,56.054,160.084
C07100=1016.565,-14.316,-106.285,165.884,56.061,160.085
C07101=1016.560,-14.565,-106.273,165.881,56.069,160.086
C07102=1016.555,-14.814,-106.261,165.878,56.076,160.086
C07103=1016.549,-15.064,-106.248,165.876,56.083,160.087
C07104=1016.544,-15.313,-106.235,165.874,56.091,160.088
C07105=1016.539,-15.564,-106.222,165.871,56.097,160.089
C07106=1016.534,-15.813,-106.211,165.868,56.105,160.090
C07107=1016.529,-16.063,-106.199,165.865,56.112,160.090
C07108=1016.523,-16.313,-106.186,165.862,56.119,160.091
C07109=1016.517,-16.562,-106.174,165.860,56.127,160.092
C07110=1016.512,-16.812,-106.161,165.857,56.135,160.093
C07111=1016.507,-17.062,-106.149,165.855,56.142,160.093
C07112=1016.502,-17.311,-106.137,165.852,56.149,160.094
C07113=1016.496,-17.561,-106.124,165.849,56.157,160.095
C07114=1016.491,-17.811,-106.113,165.847,56.164,160.095
C07115=1016.486,-18.060,-106.101,165.844,56.172,160.096
C07116=1016.480,-18.310,-106.088,165.841,56.179,160.097
C07117=1016.475,-18.559,-106.077,165.838,56.186,160.098
C07118=1016.470,-18.809,-106.065,165.836,56.194,160.098
C07119=1016.464,-19.058,-106.052,165.833,56.201,160.099
C07120=1016.459,-19.308,-106.041,165.830,56.208,160.100
C07121=1016.454,-19.558,-106.028,165.828,56.216,160.101
C07122=1016.448,-19.808,-106.015,165.825,56.223,160.101
C07123=1016.443,-20.057,-106.004,165.822,56.230,160.102
C07124=1016.438,-20.307,-105.992,165.819,56.238,160.103
C07125=1016.433,-20.556,-105.980,165.817,56.245,160.104
C07126=1016.427,-20.806,-105.967,165.814,56.252,160.104
C07127=1016.422,-21.055,-105.955,165.811,56.260,160.105
C07128=1016.416,-21.333,-105.942,165.808,56.268,160.106
C07129=1016.410,-21.609,-105.929,165.806,56.276,160.107
C07130=1016.404,-21.887,-105.916,165.802,56.284,160.107
C07131=1016.398,-22.164,-105.902,165.798,56.292,160.108
C07132=1016.393,-22.414,-105.890,165.796,56.300,160.109
C07133=1016.388,-22.663,-105.878,165.794,56.307,160.110
C07134=1016.383,-22.913,-105.866,165.791,56.314,160.110
C07135=1016.377,-23.163,-105.854,165.789,56.321,160.111
C07136=1016.372,-23.413,-105.842,165.786,56.328,160.112
C07137=1016.367,-23.662,-105.830,165.783,56.336,160.112
C07138=1016.361,-23.911,-105.818,165.780,56.343,160.113
C07139=1016.356,-24.162,-105.806,165.778,56.350,160.114
C07140=1016.351,-24.411,-105.794,165.775,56.358,160.115
C07141=1016.346,-24.661,-105.782,165.772,56.365,160.115
C07142=1016.340,-24.910,-105.770,165.769,56.372,160.116
C07143=1016.335,-25.160,-105.759,165.766,56.379,160.117
C07144=1016.329,-25.410,-105.746,165.764,56.387,160.117
C07145=1016.324,-25.659,-105.735,165.761,56.394,160.118
C07146=1016.320,-25.909,-105.722,165.758,56.401,160.119
C07147=1016.315,-26.159,-105.710,165.755,56.408,160.119
C07148=1016.309,-26.408,-105.698,165.754,56.415,160.120
C07149=1016.304,-26.658,-105.686,165.751,56.422,160.121
C07150=1016.299,-26.908,-105.675,165.748,56.430,160.122
C07151=1016.294,-27.157,-105.663,165.745,56.437,160.122
